// TwinCAT 3 PLC project PRG_B_StatesAndModes
// Title: B_StatesAndModes
// Company: RafalOS
// Author: Rafał Osajda
// ProjectVersion: 0.0.0.24
// ProgramVersion: 3.1.4024.0
// libraries:
//   B_Base, * (RafalOS)
//   Tc2_Standard, * (Beckhoff Automation GmbH)
//   Tc2_System, * (Beckhoff Automation GmbH)
//   Tc3_Module, * (Beckhoff Automation GmbH)
// project tree:
//   GVLs/ GVL_SaMConstans.TcGVL (not stored)
//   / PlcTask.TcTTO
//   POUs Compilation/ PRG_Compilation.TcPOU (not stored)
//   POUs/01_StatesAndModes/ E_SaMChangeCategory.TcDUT (not stored), E_SaMCommandChangeState.TcDUT, E_SaMCommandChangeMode.TcDUT (not stored), FB_SaMController.TcPOU, ITF_SaMController.TcIO, ITF_SaMControllerCommandChange.TcIO, ITF_SaMControllerConfigure.TcIO (not stored), ST_CommandChangeMode.TcDUT, ST_CommandChangeState.TcDUT, ST_SaMControllerConfigure.TcDUT (not stored), ST_SaMElementModes.TcDUT (not stored), ST_SaMElementStates.TcDUT (not stored)
//   POUs/02_CommandChange/ FB_CommandChange.TcPOU, ITF_CommandChange.TcIO (not stored)
//   POUs/03_CommandChangeState/ FB_CommandChangeAbort.TcPOU, FB_CommandChangeClear.TcPOU, FB_CommandChangeReset.TcPOU, FB_CommandChangeStart.TcPOU, FB_CommandChangeStop.TcPOU, FB_CommandChangeHold.TcPOU, FB_CommandChangeUnHold.TcPOU, FB_CommandChangeSuspend.TcPOU, FB_CommandChangeUnSuspend.TcPOU, FB_CommandChangeComplete.TcPOU
//   POUs/04_CommandChangeMode/ FB_CommandChangeProduction.TcPOU, FB_CommandChangeMaintenance.TcPOU, FB_CommandChangeManual.TcPOU, FB_CommandChangeWashing.TcPOU, FB_CommandChangeDiagnostics.TcPOU
//   POUs/05_SaMElement/ FB_SaMElement.TcPOU, ITF_SaMElement.TcIO
//   POUs/06_SaMElementStates/ FB_SaMElementAborting.TcPOU, FB_SaMElementAborted.TcPOU (not stored), FB_SaMElementUndefined.TcPOU (not stored), FB_SaMElementClearing.TcPOU (not stored), FB_SaMElementStopping.TcPOU (not stored), FB_SaMElementStopped.TcPOU, FB_SaMElementResseting.TcPOU, FB_SaMElementIdle.TcPOU (not stored), FB_SaMElementStarting.TcPOU, FB_SaMElementExecute.TcPOU (not stored), FB_SaMElementSuspending.TcPOU (not stored), FB_SaMElementSuspended.TcPOU, FB_SaMElementUnSuspending.TcPOU (not stored), FB_SaMElementHolding.TcPOU (not stored), FB_SaMElementHeld.TcPOU (not stored), FB_SaMElementUnHolding.TcPOU (not stored), FB_SaMElementCompleting.TcPOU (not stored), FB_SaMElementComplete.TcPOU (not stored)
//   POUs/07_SaMElementModes/ FB_SaMElementProduction.TcPOU, FB_SaMElementMaintenance.TcPOU (not stored), FB_SaMElementManual.TcPOU, FB_SaMElementNotAllowed.TcPOU (not stored), FB_SaMElementWashing.TcPOU, FB_SaMElementDiagnostics.TcPOU (not stored)

CONFIGURATION PRG_B_StatesAndModes
    RESOURCE PLC ON TwinCAT3
        TASK PlcTask(INTERVAL := T#10ms, PRIORITY := 20);
        PROGRAM PRG_Compilation WITH PlcTask : PRG_Compilation;
    END_RESOURCE
END_CONFIGURATION

// ---- POUs/01_StatesAndModes/E_SaMCommandChangeState.TcDUT
{attribute 'qualified_only'}
{attribute 'strict'}
TYPE E_SaMCommandChangeState :
(
	None			:= 0,
	Abort			:= 1,
    Clear			:= 2,
    Reset			:= 3,
    Start			:= 4,
    Stop			:= 5,
    Hold			:= 6,
    Unhold			:= 7,
    Suspend			:= 8,
    Unsuspend		:= 9,
    Complete		:= 10
);
END_TYPE

// ---- POUs/01_StatesAndModes/ST_CommandChangeMode.TcDUT
TYPE ST_CommandChangeMode :
STRUCT
	cmdChangeProduction	 	  	: FB_CommandChangeProduction;
	cmdChangeMaintenance		: FB_CommandChangeMaintenance;
	cmdChangeManual		    	: FB_CommandChangeManual;
	cmdChangeWashing		   	: FB_CommandChangeWashing;
	cmdChangeDiagnostics		: FB_CommandChangeDiagnostics;
END_STRUCT
END_TYPE

// ---- POUs/01_StatesAndModes/ST_CommandChangeState.TcDUT
TYPE ST_CommandChangeState :
STRUCT
	cmdChangeAbort		   		: FB_CommandChangeAbort;
	cmdChangeClear		   		: FB_CommandChangeClear;
	cmdChangeReset		   		: FB_CommandChangeReset;
	cmdChangeStart		   		: FB_CommandChangeStart;
	cmdChangeStop		    	: FB_CommandChangeStop;
	cmdChangeHold		    	: FB_CommandChangeHold;
	cmdChangeUnhold		  		: FB_CommandChangeUnHold;
	cmdChangeSuspend		 	: FB_CommandChangeSuspend;
	cmdChangeUnSuspend	  		: FB_CommandChangeUnSuspend;
	cmdChangeComplete		 	: FB_CommandChangeComplete;

END_STRUCT
END_TYPE

// ---- POUs/01_StatesAndModes/ITF_SaMController.TcIO
INTERFACE ITF_SaMController EXTENDS ITF_BaseControlElement, ITF_SaMControllerConfigure, ITF_SaMControllerCommandChange, ITF_BaseSaM

METHOD Execute : BOOL
VAR_INPUT
	iNumberOfCommand		: INT;
	eChangeCategory			: E_SaMChangeCategory;
END_VAR
END_METHOD

METHOD ExecuteTopElementOperationsForCurrentState : BOOL
VAR_INPUT
	itfTopElement				: ITF_BaseSaMStateMethod;
END_VAR
END_METHOD

METHOD PUBLIC ExitActivState
VAR_INPUT
END_VAR
END_METHOD

METHOD PUBLIC GetActiveModeName : ST_BaseLabel
VAR_INPUT
END_VAR
END_METHOD

METHOD PUBLIC GetActiveStateName : ST_BaseLabel
VAR_INPUT
END_VAR
END_METHOD

METHOD PUBLIC GetMode : E_BaseMachineMode
VAR_INPUT
END_VAR
END_METHOD

METHOD PUBLIC GetModeName : ST_BaseLabel
VAR_INPUT
	iNumber			: INT;
END_VAR
END_METHOD

METHOD PUBLIC GetState : E_BaseMachineState
VAR_INPUT
END_VAR
END_METHOD

METHOD GetStateName : ST_BaseLabel
VAR_INPUT
	iNumber			: INT;
END_VAR
END_METHOD

METHOD PUBLIC GetTimeStateForCurrentMode : LTIME
VAR_INPUT
	iNumber		: INT;
END_VAR
END_METHOD

METHOD PUBLIC GetTimeStateForMode : LTIME
VAR_INPUT
	iMode		: int;
	iState		: INT;
END_VAR
END_METHOD

METHOD PUBLIC GetTimeWorkForMode : LTIME
VAR_INPUT
	iMode	: INT;
END_VAR
END_METHOD

METHOD PUBLIC IncrementTimeStateAndMode
VAR_INPUT
	tInterval				: TIME := T#100MS;
END_VAR
END_METHOD

METHOD PUBLIC IsChangeModeBusy : BOOL
VAR_INPUT
END_VAR
END_METHOD

METHOD PUBLIC IsChangeModeDone : BOOL
VAR_INPUT
END_VAR
END_METHOD

METHOD PUBLIC IsChangeModeStatus : BOOL
VAR_INPUT
END_VAR
END_METHOD

METHOD PUBLIC IsChangeStateBusy : BOOL
VAR_INPUT
END_VAR
END_METHOD

METHOD PUBLIC IsChangeStateDone : BOOL
VAR_INPUT
END_VAR
END_METHOD

METHOD PUBLIC IsChangeStateStatus : BOOL
VAR_INPUT
END_VAR
END_METHOD

(*			
	RafalOS
	Rafał Osajda		25.11.2025		TC 4024.66
	Zwraca czy tryb o podanym numerze jest włączony
*)
METHOD IsModeEnabled : BOOL
VAR_INPUT
	iMode 	: INT;
END_VAR
END_METHOD

(*			
	RafalOS
	Rafał Osajda		25.11.2025		TC 4024.66
	Informacja czy zadany stan jest stanem aktualnym
*)
METHOD PUBLIC IsStateIsActual : BOOL
VAR_INPUT
	iTestState	: INT;
END_VAR
END_METHOD

METHOD PUBLIC IsStateTypeActive : BOOL
VAR_INPUT
END_VAR
END_METHOD

END_INTERFACE

// ---- POUs/01_StatesAndModes/ITF_SaMControllerCommandChange.TcIO
INTERFACE ITF_SaMControllerCommandChange

METHOD PUBLIC ChangeModeTo
VAR_INPUT
	eModeIn			: E_BaseMachineMode;
END_VAR
END_METHOD

METHOD PUBLIC ChangeStateTo
VAR_INPUT
	eStateIn			: E_BaseMachineState;
END_VAR
END_METHOD

METHOD PUBLIC GetState : E_BaseMachineState
VAR_INPUT
END_VAR
END_METHOD

METHOD IsModeEnebles : BOOL
VAR_INPUT
	eMode			: E_BaseMachineMode;
END_VAR
END_METHOD

METHOD IsPossibleExitActiveState : BOOL
VAR_INPUT
END_VAR
END_METHOD

METHOD IsPossibleExitState : BOOL
VAR_INPUT
	eMode		: E_BaseMachineMode;
END_VAR
END_METHOD

METHOD PUBLIC IsStateInModeEnabled : BOOL
VAR_INPUT
	eStateIn			: E_BaseMachineState;
END_VAR
END_METHOD

END_INTERFACE

// ---- POUs/05_SaMElement/ITF_SaMElement.TcIO
INTERFACE ITF_SaMElement EXTENDS ITF_BaseComponent

METHOD public GetNextState : E_BaseMachineState
VAR_INPUT
END_VAR
END_METHOD

METHOD GetTime : LTIME
VAR_INPUT
END_VAR
END_METHOD

METHOD PUBLIC IncrementTime
VAR_INPUT
	tInterval				: TIME := T#100MS;
END_VAR
END_METHOD

METHOD PUBLIC InvokeStateForTopElement : BOOL
VAR_INPUT
	itfTopElement		: ITF_BaseSaMStateMethod;
END_VAR
END_METHOD

METHOD PUBLIC IsActive : BOOL
VAR_INPUT
END_VAR
END_METHOD

(*			
	RafalOS
	Rafał Osajda		03.11.2025		TC 4024.66
	Zwraca czy element jest właczony w systemie
*)
METHOD PUBLIC IsEnabled : BOOL
VAR_INPUT
END_VAR
END_METHOD

METHOD PUBLIC IsStateTypeActive : BOOL
VAR_INPUT
END_VAR
END_METHOD

METHOD PUBLIC ResetTime
VAR_INPUT
END_VAR
END_METHOD

(*			
	RafalOS
	Rafał Osajda		03.11.2025		TC 4024.66
	Ustawia czy dane element jest aktywny
*)
METHOD PUBLIC SetActive
VAR_INPUT
	bIN			: BOOL;
END_VAR
END_METHOD

(*			
	RafalOS
	Rafał Osajda		03.11.2025		TC 4024.66
	Ustawie czy element jest włączony w systemie
*)
METHOD PUBLIC SetEnabled
VAR_INPUT
	bIN			: BOOL;
END_VAR
END_METHOD

END_INTERFACE

// ---- POUs/01_StatesAndModes/FB_SaMController.TcPOU
(*			
	RafalOS
	Rafał Osajda		30.10.2025		TC 4024.66
	Główny FB do zarządzania stanami i trybami pracy
*)
FUNCTION_BLOCK FB_SaMController EXTENDS FB_BaseControlElement IMPLEMENTS ITF_SaMController
VAR
(*	Polecenia zmiany stany	*)	
	stCmdStates					: ST_CommandChangeState;
	arrcmdStates				: ARRAY [1..GVL_SaMConstans.NUMBER_OF_COMMAND_CHANGE_STATES] OF ITF_CommandChange;
(*	Polecenia zmiany trybu	*)
	stCmdModes					: ST_CommandChangeMode;
	arrcmdModes					: ARRAY [1..GVL_SaMConstans.NUMBER_OF_COMMAND_CHANGE_MODES] OF ITF_CommandChange;
(*	Stany	*)
	arrstStates					: ARRAY [0..GVL_SaMConstans.NUMBER_OF_MODES] OF ST_SaMElementStates;
(*	Tryby	*)
	stModes						: ST_SaMElementModes;
(*	Przypisane stany do trybów	*)
	arrStatesInModes			: ARRAY [0..GVL_SaMConstans.NUMBER_OF_MODES] OF ARRAY [0..GVL_SaMConstans.NUMBER_OF_STATES] OF ITF_SaMElement;
	arrModes					: ARRAY [0..GVL_SaMConstans.NUMBER_OF_MODES] OF ITF_SaMElement;
(*	Referencja do tablicy stanów aktywnego trybu	*)
	refarrStatesForActiveMode	: REFERENCE TO ARRAY [0..GVL_SaMConstans.NUMBER_OF_STATES] OF ITF_SaMElement;
(*	Jakie trybu są aktywne	*)
	arrModeEnable				: ARRAY [0..GVL_SaMConstans.NUMBER_OF_MODES] OF BOOL;
(*	Jakie stany są aktywne w trybie	*)
	arrStateEnableInMode		: ARRAY [0..GVL_SaMConstans.NUMBER_OF_MODES] OF ARRAY [0..GVL_SaMConstans.NUMBER_OF_STATES] OF BOOL;
(*	W jakich stanach można przejść do innego trybu	*)
	arrModeTransitionEnableInState	: ARRAY [0..GVL_SaMConstans.NUMBER_OF_MODES] OF ARRAY [0..GVL_SaMConstans.NUMBER_OF_STATES] OF BOOL;
(*	Polecenia zmiany	*)
	cmdChangeMode				: FB_BaseCommand;
	cmdChangeState				: FB_BaseCommand;
(*	Zmienne		*)
	eState						: E_BaseMachineState;	//aktualny stan
	eMode						: E_BaseMachineMode;	//aktualny tryb
	eNewState					: E_BaseMachineState;	//Nowy stan
	ePrevState					: E_BaseMachineState;	//poprzedni stan
	eNewMode					: E_BaseMachineMode;	//nowy tryb
	ePrevMode					: E_BaseMachineMode;	//poprzedni tryb
END_VAR

(*			
	RafalOS
	Rafał Osajda		04.11.2025		TC 4024.66
	cykl zmiany trybu
*)
METHOD PRIVATE ChangeModeCycle : BOOL
VAR_INPUT
END_VAR
CASE THIS^.cmdChangeMode.GetStep () OF
	0	:
		THIS^.arrModes [THIS^.eMode].SetActive (bIN := FALSE);
		THIS^.ePrevMode			:= THIS^.eMode;
		THIS^.eMode				:= THIS^.eNewMode;
		THIS^.arrModes [THIS^.eMode].SetActive (bIN := TRUE);
		THIS^.refarrStatesForActiveMode	REF= THIS^.arrStatesInModes [THIS^.eMode];
		THIS^.cmdChangeMode.SetStepAsFinal ();
END_CASE
THIS^.cmdChangeMode.TestingLastCycle ();
END_METHOD

METHOD PUBLIC ChangeModeTo
VAR_INPUT
	eModeIn			: E_BaseMachineMode;
END_VAR
THIS^.eNewMode			:= eModeIn;
THIS^.cmdChangeMode.Execute ();
END_METHOD

(*			
	RafalOS
	Rafał Osajda		04.11.2025		TC 4024.66
	cykl zmiany stanu
*)
METHOD PRIVATE ChangeStateCycle : BOOL
VAR_INPUT
END_VAR
CASE THIS^.cmdChangeState.GetStep () OF
	0	:
		THIS^.refarrStatesForActiveMode [THIS^.eState].SetActive (bIN := FALSE);
		THIS^.ePrevState		:= THIS^.eState;
		THIS^.eState			:= THIS^.eNewState;
		THIS^.refarrStatesForActiveMode [THIS^.eState].SetActive (bIN := TRUE);
		THIS^.cmdChangeState.SetStepAsFinal ();
END_CASE
THIS^.cmdChangeState.TestingLastCycle ();
END_METHOD

METHOD PUBLIC ChangeStateTo
VAR_INPUT
	eStateIn			: E_BaseMachineState;
END_VAR
THIS^.eNewState			:= eStateIn;
THIS^.cmdChangeState.Execute ();
END_METHOD

(*			
	RafalOS
	Rafał Osajda		03.11.2025		TC 4024.66
	Obsługa zmiany stanów i trybów 
*)
METHOD Execute : BOOL
VAR_INPUT
	iNumberOfCommand		: INT;
	eChangeCategory			: E_SaMChangeCategory;
END_VAR
CASE eChangeCategory OF
	E_SaMChangeCategory.eState	:
		THIS^.arrcmdStates [iNumberOfCommand].Execute (iNumberOfCommand	:= iNumberOfCommand);
	E_SaMChangeCategory.eMode	:
		THIS^.arrcmdModes [iNumberOfCommand].Execute (iNumberOfCommand	:= iNumberOfCommand);
END_CASE
END_METHOD

(*			
	RafalOS
	Rafał Osajda		27.03.2025		TC 4024.66
	Obsluga bledow sprawdzanie czy jakis blad sie nei pojawil i ustawienie stanu lub wylaczenie
*)
METHOD PUBLIC ExecuteEveryCycle_Error
VAR_INPUT
END_VAR
SUPER^.ExecuteEveryCycle_Error ();
END_METHOD

(*			
	RafalOS
	Rafał Osajda		27.03.2025		TC 4024.66
	Wywolanie co cykl operacji 
*)
METHOD PUBLIC ExecuteEveryCycle_Operation
VAR_INPUT
END_VAR
SUPER^.ExecuteEveryCycle_Operation ();

IF (THIS^.cmdChangeMode.OperationExecute ()) THEN
	THIS^.cmdChangeMode.Operation (bIN := THIS^.ChangeModeCycle ());
END_IF

IF (THIS^.cmdChangeState.OperationExecute ()) THEN
	THIS^.cmdChangeState.Operation (bIN := THIS^.ChangeStateCycle ());
END_IF
END_METHOD

(*			
	RafalOS
	Rafał Osajda		27.03.2025		TC 4024.66
	Aktualizacja flag 
*)
METHOD PUBLIC ExecuteEveryCycle_Status
VAR_INST
END_VAR
SUPER^.ExecuteEveryCycle_Status ();
END_METHOD

(*			
	RafalOS
	Rafał Osajda		27.03.2025		TC 4024.66
	Testowanie czy nei pojawil sie jakis rozkaz i uruchomienie odpowiednich operacji
*)
METHOD PUBLIC ExecuteEveryCycle_Test
VAR_INPUT
END_VAR
SUPER^.ExecuteEveryCycle_Test ();

THIS^.cmdChangeMode.Test ();
THIS^.cmdChangeState.Test ();
END_METHOD

METHOD ExecuteTopElementOperationsForCurrentState : BOOL
VAR_INPUT
	itfTopElement				: ITF_BaseSaMStateMethod;
END_VAR
ExecuteTopElementOperationsForCurrentState := THIS^.refarrStatesForActiveMode [THIS^.eState].InvokeStateForTopElement (itfTopElement := itfTopElement);
END_METHOD

(*			
	RafalOS
	Rafał Osajda		04.11.2025		TC 4024.66
	Wywołanie odpowiednie metody tak by wyjśc z aktualnego stanu aktywnego 
*)
METHOD PUBLIC ExitActivState
VAR_INPUT
END_VAR
THIS^.ChangeStateTo (eStateIn := THIS^.refarrStatesForActiveMode [THIS^.eState].GetNextState ());
END_METHOD

METHOD FB_init : BOOL
VAR_INPUT
	bInitRetains : BOOL; // if TRUE, the retain variables are initialized (warm start / cold start)
	bInCopyCode : BOOL;  // if TRUE, the instance afterwards gets moved into the copy code (online change)
END_VAR
THIS^.SetText (eLocation := E_BaseLocation.pl, wsDescription := "SaM Controller");
THIS^.SetText (eLocation := E_BaseLocation.en, wsDescription := "SaM Controller");
THIS^.SetText (eLocation := E_BaseLocation.de, wsDescription := "SaM Controller");
THIS^.SetName (stName := THIS^.GetTexts ());

THIS^.Initialization_AddStates ();
THIS^.Initialization_AddModes ();

THIS^.Initialization_AddCommandChangeState ();
THIS^.Initialization_AddCommandChangeModes ();

THIS^.Initialization_StateEnabledInMode ();
THIS^.Initialization_ModeTransitionEnabledInState ();
THIS^.Initialization_ModeEnabled ();
END_METHOD

METHOD PUBLIC GetActiveModeName : ST_BaseLabel
VAR_INPUT
END_VAR
GetActiveModeName := THIS^.GetModeName (iNumber := THIS^.eMode);
END_METHOD

METHOD PUBLIC GetActiveStateName : ST_BaseLabel
VAR_INPUT
END_VAR
GetActiveStateName := THIS^.GetStateName (iNumber := THIS^.eState);
END_METHOD

METHOD PUBLIC GetMode : E_BaseMachineMode
VAR_INPUT
END_VAR
GetMode			:= THIS^.eMode;
END_METHOD

METHOD PUBLIC GetModeName : ST_BaseLabel
VAR_INPUT
	iNumber			: INT;
END_VAR
GetModeName := THIS^.arrModes [iNumber].GetName ();
END_METHOD

METHOD PUBLIC GetState : E_BaseMachineState
VAR_INPUT
END_VAR
GetState			:= THIS^.eState;
END_METHOD

METHOD GetStateName : ST_BaseLabel
VAR_INPUT
	iNumber			: INT;
END_VAR
GetStateName := THIS^.arrStatesInModes [THIS^.eMode][iNumber].GetName ();
END_METHOD

METHOD PUBLIC GetTimeStateForCurrentMode : LTIME
VAR_INPUT
	iNumber		: INT;
END_VAR
GetTimeStateForCurrentMode := this^.refarrStatesForActiveMode [iNumber].GetTime ();
END_METHOD

METHOD PUBLIC GetTimeStateForMode : LTIME
VAR_INPUT
	iMode		: INT;
	iState		: INT;
END_VAR
GetTimeStateForMode := THIS^.arrStatesInModes [iMode][iState].GetTime ();
END_METHOD

METHOD PUBLIC GetTimeWorkForMode : LTIME
VAR_INPUT
	iMode	: INT;
END_VAR
GetTimeWorkForMode := THIS^.arrModes [iMode].GetTime ();
END_METHOD

METHOD PUBLIC IncrementTimeStateAndMode
VAR_INPUT
	tInterval				: TIME := T#100MS;
END_VAR
THIS^.refarrStatesForActiveMode [THIS^.eState].IncrementTime (tInterval := tInterval);
THIS^.arrModes [THIS^.eMode].IncrementTime (tInterval := tInterval);
END_METHOD

METHOD PRIVATE Initialization_AddCommandChangeModes : BOOL
VAR_INPUT
END_VAR

THIS^.arrcmdModes [E_SaMCommandChangeMode.Production]	:= THIS^.stCmdModes.cmdChangeProduction;
THIS^.AddComponent (itfComponent 	:= THIS^.stCmdModes.cmdChangeProduction);
THIS^.stCmdModes.cmdChangeProduction.LinkSaMCotroller (itfSaMController	:= THIS^);

THIS^.arrcmdModes [E_SaMCommandChangeMode.Maintenance]	:= THIS^.stCmdModes.cmdChangeMaintenance;
THIS^.AddComponent (itfComponent 	:= THIS^.stCmdModes.cmdChangeMaintenance);
THIS^.stCmdModes.cmdChangeMaintenance.LinkSaMCotroller (itfSaMController	:= THIS^);

THIS^.arrcmdModes [E_SaMCommandChangeMode.Manual]		:= THIS^.stCmdModes.cmdChangeManual;
THIS^.AddComponent (itfComponent 	:= THIS^.stCmdModes.cmdChangeManual);
THIS^.stCmdModes.cmdChangeManual.LinkSaMCotroller (itfSaMController	:= THIS^);

THIS^.arrcmdModes [E_SaMCommandChangeMode.Washing]		:= THIS^.stCmdModes.cmdChangeWashing;
THIS^.AddComponent (itfComponent 	:= THIS^.stCmdModes.cmdChangeWashing);
THIS^.stCmdModes.cmdChangeWashing.LinkSaMCotroller (itfSaMController	:= THIS^);

THIS^.arrcmdModes [E_SaMCommandChangeMode.Diagnostisc]	:= THIS^.stCmdModes.cmdChangeDiagnostics;
THIS^.AddComponent (itfComponent 	:= THIS^.stCmdModes.cmdChangeDiagnostics);
THIS^.stCmdModes.cmdChangeDiagnostics.LinkSaMCotroller (itfSaMController	:= THIS^);
END_METHOD

METHOD PRIVATE Initialization_AddCommandChangeState : BOOL
VAR_INPUT
END_VAR
THIS^.arrcmdStates [E_SaMCommandChangeState.Abort]	:= THIS^.stCmdStates.cmdChangeAbort;
THIS^.AddComponent (itfComponent 	:= THIS^.stCmdStates.cmdChangeAbort);
THIS^.stCmdStates.cmdChangeAbort.LinkSaMCotroller (itfSaMController	:= THIS^);

THIS^.arrcmdStates [E_SaMCommandChangeState.Clear]	:= THIS^.stCmdStates.cmdChangeClear;
THIS^.AddComponent (itfComponent 	:= THIS^.stCmdStates.cmdChangeClear);
THIS^.stCmdStates.cmdChangeClear.LinkSaMCotroller (itfSaMController	:= THIS^);

THIS^.arrcmdStates [E_SaMCommandChangeState.Reset]	:= THIS^.stCmdStates.cmdChangeReset;
THIS^.AddComponent (itfComponent 	:= THIS^.stCmdStates.cmdChangeReset);
THIS^.stCmdStates.cmdChangeReset.LinkSaMCotroller (itfSaMController	:= THIS^);

THIS^.arrcmdStates [E_SaMCommandChangeState.Start]	:= THIS^.stCmdStates.cmdChangeStart;
THIS^.AddComponent (itfComponent 	:= THIS^.stCmdStates.cmdChangeStart);
THIS^.stCmdStates.cmdChangeStart.LinkSaMCotroller (itfSaMController	:= THIS^);

THIS^.arrcmdStates [E_SaMCommandChangeState.Stop]	:= THIS^.stCmdStates.cmdChangeStop;
THIS^.AddComponent (itfComponent 	:= THIS^.stCmdStates.cmdChangeStop);
THIS^.stCmdStates.cmdChangeStop.LinkSaMCotroller (itfSaMController	:= THIS^);

THIS^.arrcmdStates [E_SaMCommandChangeState.Hold]	:= THIS^.stCmdStates.cmdChangeHold;
THIS^.AddComponent (itfComponent 	:= THIS^.stCmdStates.cmdChangeHold);
THIS^.stCmdStates.cmdChangeHold.LinkSaMCotroller (itfSaMController	:= THIS^);

THIS^.arrcmdStates [E_SaMCommandChangeState.Unhold]	:= THIS^.stCmdStates.cmdChangeUnhold;
THIS^.AddComponent (itfComponent 	:= THIS^.stCmdStates.cmdChangeUnhold);
THIS^.stCmdStates.cmdChangeUnhold.LinkSaMCotroller (itfSaMController	:= THIS^);

THIS^.arrcmdStates [E_SaMCommandChangeState.Suspend]:= THIS^.stCmdStates.cmdChangeSuspend;
THIS^.AddComponent (itfComponent 	:= THIS^.stCmdStates.cmdChangeSuspend);
THIS^.stCmdStates.cmdChangeSuspend.LinkSaMCotroller (itfSaMController	:= THIS^);

THIS^.arrcmdStates [E_SaMCommandChangeState.Unsuspend]	:= THIS^.stCmdStates.cmdChangeUnSuspend;
THIS^.AddComponent (itfComponent 	:= THIS^.stCmdStates.cmdChangeUnSuspend);
THIS^.stCmdStates.cmdChangeUnSuspend.LinkSaMCotroller (itfSaMController	:= THIS^);

THIS^.arrcmdStates [E_SaMCommandChangeState.Complete]	:= THIS^.stCmdStates.cmdChangeComplete;
THIS^.AddComponent (itfComponent 	:= THIS^.stCmdStates.cmdChangeComplete);
THIS^.stCmdStates.cmdChangeComplete.LinkSaMCotroller (itfSaMController	:= THIS^);
END_METHOD

METHOD PRIVATE Initialization_AddModes : BOOL
VAR_INPUT
END_VAR
THIS^.arrModes [E_BaseMachineMode.NotAllowed]	:= THIS^.stModes.fbUndefined;
THIS^.AddComponent (itfComponent	:= THIS^.stModes.fbUndefined);
THIS^.arrModes [E_BaseMachineMode.Production]	:= THIS^.stModes.fbProduction;
THIS^.AddComponent (itfComponent	:= THIS^.stModes.fbProduction);
THIS^.arrModes [E_BaseMachineMode.Maintenance]	:= THIS^.stModes.fbMaintenance;
THIS^.AddComponent (itfComponent	:= THIS^.stModes.fbMaintenance);
THIS^.arrModes [E_BaseMachineMode.Manual]	:= THIS^.stModes.fbManual;
THIS^.AddComponent (itfComponent	:= THIS^.stModes.fbManual);
THIS^.arrModes [E_BaseMachineMode.Washing]	:= THIS^.stModes.fbWashing;
THIS^.AddComponent (itfComponent	:= THIS^.stModes.fbWashing);
THIS^.arrModes [E_BaseMachineMode.Diagnostics]	:= THIS^.stModes.fbDiagnostics;
THIS^.AddComponent (itfComponent	:= THIS^.stModes.fbDiagnostics);
END_METHOD

METHOD PRIVATE Initialization_AddStates : BOOL
VAR_INPUT
END_VAR

VAR
	iI: INT;
END_VAR
FOR iI := 0 TO GVL_SaMConstans.NUMBER_OF_MODES DO
	THIS^.arrStatesInModes [iI][E_BaseMachineState.Undefined] 		:= THIS^.arrstStates [iI].fbUndefined;
	THIS^.arrStatesInModes [iI][E_BaseMachineState.Aborting] 		:= THIS^.arrstStates [iI].fbAborting;
	THIS^.arrStatesInModes [iI][E_BaseMachineState.Aborted] 		:= THIS^.arrstStates [iI].fbAborted;
	THIS^.arrStatesInModes [iI][E_BaseMachineState.Clearing] 		:= THIS^.arrstStates [iI].fbClearing;
	THIS^.arrStatesInModes [iI][E_BaseMachineState.Stopping] 		:= THIS^.arrstStates [iI].fbStopping;
	THIS^.arrStatesInModes [iI][E_BaseMachineState.Stopped] 		:= THIS^.arrstStates [iI].fbStopped;
	THIS^.arrStatesInModes [iI][E_BaseMachineState.Resetting] 		:= THIS^.arrstStates [iI].fbResetting;
	THIS^.arrStatesInModes [iI][E_BaseMachineState.Idle] 			:= THIS^.arrstStates [iI].fbIdle;
	THIS^.arrStatesInModes [iI][E_BaseMachineState.Starting] 		:= THIS^.arrstStates [iI].fbStarting;
	THIS^.arrStatesInModes [iI][E_BaseMachineState.Execute] 		:= THIS^.arrstStates [iI].fbExecute;
	THIS^.arrStatesInModes [iI][E_BaseMachineState.Suspending]	 	:= THIS^.arrstStates [iI].fbSuspending;
	THIS^.arrStatesInModes [iI][E_BaseMachineState.Suspended] 		:= THIS^.arrstStates [iI].fbSuspended;
	THIS^.arrStatesInModes [iI][E_BaseMachineState.Unsuspending]	:= THIS^.arrstStates [iI].fbUnsuspending;
	THIS^.arrStatesInModes [iI][E_BaseMachineState.Holding] 		:= THIS^.arrstStates [iI].fbHolding;
	THIS^.arrStatesInModes [iI][E_BaseMachineState.Held] 			:= THIS^.arrstStates [iI].fbHeld;
	THIS^.arrStatesInModes [iI][E_BaseMachineState.Unholding] 		:= THIS^.arrstStates [iI].fbUnholding;
	THIS^.arrStatesInModes [iI][E_BaseMachineState.Completing] 	:= THIS^.arrstStates [iI].fbCompleting;
	THIS^.arrStatesInModes [iI][E_BaseMachineState.Complete] 		:= THIS^.arrstStates [iI].fbComplete;
	THIS^.AddComponent (itfComponent 	:= THIS^.arrstStates [iI].fbUndefined);
	THIS^.AddComponent (itfComponent 	:= THIS^.arrstStates [iI].fbAborting);
	THIS^.AddComponent (itfComponent 	:= THIS^.arrstStates [iI].fbAborted);
	THIS^.AddComponent (itfComponent 	:= THIS^.arrstStates [iI].fbClearing);
	THIS^.AddComponent (itfComponent 	:= THIS^.arrstStates [iI].fbStopping);
	THIS^.AddComponent (itfComponent 	:= THIS^.arrstStates [iI].fbStopped);
	THIS^.AddComponent (itfComponent 	:= THIS^.arrstStates [iI].fbResetting);
	THIS^.AddComponent (itfComponent 	:= THIS^.arrstStates [iI].fbIdle);
	THIS^.AddComponent (itfComponent 	:= THIS^.arrstStates [iI].fbStarting);
	THIS^.AddComponent (itfComponent 	:= THIS^.arrstStates [iI].fbExecute);
	THIS^.AddComponent (itfComponent 	:= THIS^.arrstStates [iI].fbSuspending);
	THIS^.AddComponent (itfComponent 	:= THIS^.arrstStates [iI].fbSuspended);
	THIS^.AddComponent (itfComponent 	:= THIS^.arrstStates [iI].fbUnsuspending);
	THIS^.AddComponent (itfComponent 	:= THIS^.arrstStates [iI].fbHolding);
	THIS^.AddComponent (itfComponent 	:= THIS^.arrstStates [iI].fbHeld);
	THIS^.AddComponent (itfComponent 	:= THIS^.arrstStates [iI].fbUnholding);
	THIS^.AddComponent (itfComponent 	:= THIS^.arrstStates [iI].fbCompleting);
	THIS^.AddComponent (itfComponent 	:= THIS^.arrstStates [iI].fbComplete);
END_FOR
END_METHOD

(*			
	RafalOS
	Rafał Osajda		03.11.2025		TC 4024.66
	Przepisuje ustawiony stan Enebled z elementu i zapisuje go do tablisy trybów
*)
METHOD PRIVATE Initialization_CopeEnabledMode
VAR
	iI: INT;
END_VAR
FOR iI := 0 TO GVL_SaMConstans.NUMBER_OF_MODES DO
	IF (THIS^.arrModes [iI] <> 0) THEN
		THIS^.arrModeEnable [iI]	:= THIS^.arrModes [iI].IsEnabled ();
	END_IF
END_FOR
END_METHOD

(*			
	RafalOS
	Rafał Osajda		03.11.2025		TC 4024.66
	Przepisuje ustawiony stan Enebled z elementu i zapisuje go do tablisy stanów w trybach
*)
METHOD PRIVATE Initialization_CopeEnabledStateToMode
VAR_INPUT
	eMode			: E_BaseMachineMode;
END_VAR

VAR
	iI: INT;
END_VAR
FOR iI := 0 TO GVL_SaMConstans.NUMBER_OF_STATES DO
	IF (THIS^.arrStatesInModes [eMode][iI] <> 0) THEN
		THIS^.arrStateEnableInMode [eMode][iI]	:= THIS^.arrStatesInModes [eMode][iI].IsEnabled ();
	END_IF
END_FOR
END_METHOD

(*			
	RafalOS
	Rafał Osajda		03.11.2025		TC 4024.66
	Inicjalizacja jakie tryby są właczony
*)
METHOD PRIVATE Initialization_ModeEnabled
VAR_INPUT
END_VAR
THIS^.stModes.fbUndefined.SetEnabled (bIN	:= TRUE);
THIS^.stModes.fbProduction.SetEnabled (bIN	:= TRUE);
THIS^.stModes.fbMaintenance.SetEnabled (bIN	:= TRUE);
THIS^.stModes.fbManual.SetEnabled (bIN	:= TRUE);
THIS^.stModes.fbWashing.SetEnabled (bIN	:= TRUE);
THIS^.stModes.fbDiagnostics.SetEnabled (bIN	:= TRUE);
THIS^.Initialization_CopeEnabledMode ();
END_METHOD

(*			
	RafalOS
	Rafał Osajda		03.11.2025		TC 4024.66
	Ustawienie w jakim stanie trybu mozemy zmieniać tryby
*)
METHOD PRIVATE Initialization_ModeTransitionEnabledInState
VAR_INPUT
END_VAR
THIS^.arrModeTransitionEnableInState [E_BaseMachineMode.NotAllowed][E_BaseMachineState.Undefined]		:= TRUE;
THIS^.arrModeTransitionEnableInState [E_BaseMachineMode.Production][E_BaseMachineState.Undefined]		:= TRUE;
THIS^.arrModeTransitionEnableInState [E_BaseMachineMode.Maintenance][E_BaseMachineState.Undefined]		:= TRUE;
THIS^.arrModeTransitionEnableInState [E_BaseMachineMode.Manual][E_BaseMachineState.Undefined]			:= TRUE;
THIS^.arrModeTransitionEnableInState [E_BaseMachineMode.Washing][E_BaseMachineState.Undefined]		:= TRUE;
THIS^.arrModeTransitionEnableInState [E_BaseMachineMode.Diagnostics][E_BaseMachineState.Undefined]	:= TRUE;

THIS^.arrModeTransitionEnableInState [E_BaseMachineMode.NotAllowed][E_BaseMachineState.Aborted]		:= TRUE;
THIS^.arrModeTransitionEnableInState [E_BaseMachineMode.Production][E_BaseMachineState.Aborted]		:= TRUE;
THIS^.arrModeTransitionEnableInState [E_BaseMachineMode.Maintenance][E_BaseMachineState.Aborted]		:= TRUE;
THIS^.arrModeTransitionEnableInState [E_BaseMachineMode.Manual][E_BaseMachineState.Aborted]			:= TRUE;
THIS^.arrModeTransitionEnableInState [E_BaseMachineMode.Washing][E_BaseMachineState.Aborted]			:= TRUE;
THIS^.arrModeTransitionEnableInState [E_BaseMachineMode.Diagnostics][E_BaseMachineState.Aborted]		:= TRUE;

THIS^.arrModeTransitionEnableInState [E_BaseMachineMode.NotAllowed][E_BaseMachineState.Stopped]		:= TRUE;
THIS^.arrModeTransitionEnableInState [E_BaseMachineMode.Production][E_BaseMachineState.Stopped]		:= TRUE;
THIS^.arrModeTransitionEnableInState [E_BaseMachineMode.Maintenance][E_BaseMachineState.Stopped]		:= TRUE;
THIS^.arrModeTransitionEnableInState [E_BaseMachineMode.Manual][E_BaseMachineState.Stopped]			:= TRUE;
THIS^.arrModeTransitionEnableInState [E_BaseMachineMode.Washing][E_BaseMachineState.Stopped]			:= TRUE;
THIS^.arrModeTransitionEnableInState [E_BaseMachineMode.Diagnostics][E_BaseMachineState.Stopped]		:= TRUE;
END_METHOD

(*			
	RafalOS
	Rafał Osajda		03.11.2025		TC 4024.66
	Ustawienie jakie stany sa włączone w jakim stanie
*)
METHOD PRIVATE Initialization_StateEnabledInMode
VAR_INPUT
END_VAR
THIS^.arrstStates [E_BaseMachineMode.NotAllowed].fbUndefined.SetEnabled (bIN		:= TRUE);
THIS^.arrstStates [E_BaseMachineMode.NotAllowed].fbAborting.SetEnabled (bIN		:= FALSE);
THIS^.arrstStates [E_BaseMachineMode.NotAllowed].fbAborted.SetEnabled (bIN			:= FALSE);
THIS^.arrstStates [E_BaseMachineMode.NotAllowed].fbClearing.SetEnabled (bIN 		:= FALSE);
THIS^.arrstStates [E_BaseMachineMode.NotAllowed].fbStopping.SetEnabled (bIN 		:= FALSE);
THIS^.arrstStates [E_BaseMachineMode.NotAllowed].fbStopped.SetEnabled (bIN 		:= FALSE);
THIS^.arrstStates [E_BaseMachineMode.NotAllowed].fbResetting.SetEnabled (bIN 		:= FALSE);
THIS^.arrstStates [E_BaseMachineMode.NotAllowed].fbIdle.SetEnabled (bIN 			:= FALSE);
THIS^.arrstStates [E_BaseMachineMode.NotAllowed].fbStarting.SetEnabled (bIN 		:= FALSE);
THIS^.arrstStates [E_BaseMachineMode.NotAllowed].fbExecute.SetEnabled (bIN 		:= FALSE);
THIS^.arrstStates [E_BaseMachineMode.NotAllowed].fbSuspending.SetEnabled (bIN 		:= FALSE);
THIS^.arrstStates [E_BaseMachineMode.NotAllowed].fbSuspended.SetEnabled (bIN 		:= FALSE);
THIS^.arrstStates [E_BaseMachineMode.NotAllowed].fbUnsuspending.SetEnabled (bIN	:= FALSE);
THIS^.arrstStates [E_BaseMachineMode.NotAllowed].fbHolding.SetEnabled (bIN 		:= FALSE);
THIS^.arrstStates [E_BaseMachineMode.NotAllowed].fbHeld.SetEnabled (bIN 			:= FALSE);
THIS^.arrstStates [E_BaseMachineMode.NotAllowed].fbUnholding.SetEnabled (bIN 		:= FALSE);
THIS^.arrstStates [E_BaseMachineMode.NotAllowed].fbCompleting.SetEnabled (bIN 		:= FALSE);
THIS^.arrstStates [E_BaseMachineMode.NotAllowed].fbComplete.SetEnabled (bIN 		:= FALSE);
THIS^.Initialization_CopeEnabledStateToMode (eMode	:= E_BaseMachineMode.NotAllowed);


THIS^.arrstStates [E_BaseMachineMode.Production].fbUndefined.SetEnabled (bIN		:= TRUE);
THIS^.arrstStates [E_BaseMachineMode.Production].fbAborting.SetEnabled (bIN		:= TRUE);
THIS^.arrstStates [E_BaseMachineMode.Production].fbAborted.SetEnabled (bIN			:= TRUE);
THIS^.arrstStates [E_BaseMachineMode.Production].fbClearing.SetEnabled (bIN 		:= TRUE);
THIS^.arrstStates [E_BaseMachineMode.Production].fbStopping.SetEnabled (bIN 		:= TRUE);
THIS^.arrstStates [E_BaseMachineMode.Production].fbStopped.SetEnabled (bIN 		:= TRUE);
THIS^.arrstStates [E_BaseMachineMode.Production].fbResetting.SetEnabled (bIN 		:= TRUE);
THIS^.arrstStates [E_BaseMachineMode.Production].fbIdle.SetEnabled (bIN 			:= TRUE);
THIS^.arrstStates [E_BaseMachineMode.Production].fbStarting.SetEnabled (bIN 		:= TRUE);
THIS^.arrstStates [E_BaseMachineMode.Production].fbExecute.SetEnabled (bIN 		:= TRUE);
THIS^.arrstStates [E_BaseMachineMode.Production].fbSuspending.SetEnabled (bIN 		:= TRUE);
THIS^.arrstStates [E_BaseMachineMode.Production].fbSuspended.SetEnabled (bIN 		:= TRUE);
THIS^.arrstStates [E_BaseMachineMode.Production].fbUnsuspending.SetEnabled (bIN	:= TRUE);
THIS^.arrstStates [E_BaseMachineMode.Production].fbHolding.SetEnabled (bIN 		:= TRUE);
THIS^.arrstStates [E_BaseMachineMode.Production].fbHeld.SetEnabled (bIN 			:= TRUE);
THIS^.arrstStates [E_BaseMachineMode.Production].fbUnholding.SetEnabled (bIN 		:= TRUE);
THIS^.arrstStates [E_BaseMachineMode.Production].fbCompleting.SetEnabled (bIN 		:= TRUE);
THIS^.arrstStates [E_BaseMachineMode.Production].fbComplete.SetEnabled (bIN 		:= TRUE);
THIS^.Initialization_CopeEnabledStateToMode (eMode	:= E_BaseMachineMode.Production);

THIS^.arrstStates [E_BaseMachineMode.Maintenance].fbUndefined.SetEnabled (bIN		:= TRUE);
THIS^.arrstStates [E_BaseMachineMode.Maintenance].fbAborting.SetEnabled (bIN			:= TRUE);
THIS^.arrstStates [E_BaseMachineMode.Maintenance].fbAborted.SetEnabled (bIN			:= TRUE);
THIS^.arrstStates [E_BaseMachineMode.Maintenance].fbClearing.SetEnabled (bIN 		:= TRUE);
THIS^.arrstStates [E_BaseMachineMode.Maintenance].fbStopping.SetEnabled (bIN 		:= TRUE);
THIS^.arrstStates [E_BaseMachineMode.Maintenance].fbStopped.SetEnabled (bIN 			:= TRUE);
THIS^.arrstStates [E_BaseMachineMode.Maintenance].fbResetting.SetEnabled (bIN 		:= TRUE);
THIS^.arrstStates [E_BaseMachineMode.Maintenance].fbIdle.SetEnabled (bIN 			:= TRUE);
THIS^.arrstStates [E_BaseMachineMode.Maintenance].fbStarting.SetEnabled (bIN 		:= TRUE);
THIS^.arrstStates [E_BaseMachineMode.Maintenance].fbExecute.SetEnabled (bIN 			:= TRUE);
THIS^.arrstStates [E_BaseMachineMode.Maintenance].fbSuspending.SetEnabled (bIN 		:= FALSE);
THIS^.arrstStates [E_BaseMachineMode.Maintenance].fbSuspended.SetEnabled (bIN 		:= FALSE);
THIS^.arrstStates [E_BaseMachineMode.Maintenance].fbUnsuspending.SetEnabled (bIN		:= FALSE);
THIS^.arrstStates [E_BaseMachineMode.Maintenance].fbHolding.SetEnabled (bIN 			:= FALSE);
THIS^.arrstStates [E_BaseMachineMode.Maintenance].fbHeld.SetEnabled (bIN 			:= FALSE);
THIS^.arrstStates [E_BaseMachineMode.Maintenance].fbUnholding.SetEnabled (bIN 		:= FALSE);
THIS^.arrstStates [E_BaseMachineMode.Maintenance].fbCompleting.SetEnabled (bIN 		:= FALSE);
THIS^.arrstStates [E_BaseMachineMode.Maintenance].fbComplete.SetEnabled (bIN 		:= FALSE);
THIS^.Initialization_CopeEnabledStateToMode (eMode	:= E_BaseMachineMode.Maintenance);

THIS^.arrstStates [E_BaseMachineMode.Manual].fbUndefined.SetEnabled (bIN			:= TRUE);
THIS^.arrstStates [E_BaseMachineMode.Manual].fbAborting.SetEnabled (bIN			:= TRUE);
THIS^.arrstStates [E_BaseMachineMode.Manual].fbAborted.SetEnabled (bIN				:= TRUE);
THIS^.arrstStates [E_BaseMachineMode.Manual].fbClearing.SetEnabled (bIN 			:= TRUE);
THIS^.arrstStates [E_BaseMachineMode.Manual].fbStopping.SetEnabled (bIN 			:= TRUE);
THIS^.arrstStates [E_BaseMachineMode.Manual].fbStopped.SetEnabled (bIN 			:= TRUE);
THIS^.arrstStates [E_BaseMachineMode.Manual].fbResetting.SetEnabled (bIN 			:= TRUE);
THIS^.arrstStates [E_BaseMachineMode.Manual].fbIdle.SetEnabled (bIN 				:= TRUE);
THIS^.arrstStates [E_BaseMachineMode.Manual].fbStarting.SetEnabled (bIN 			:= TRUE);
THIS^.arrstStates [E_BaseMachineMode.Manual].fbExecute.SetEnabled (bIN 			:= TRUE);
THIS^.arrstStates [E_BaseMachineMode.Manual].fbSuspending.SetEnabled (bIN 			:= TRUE);
THIS^.arrstStates [E_BaseMachineMode.Manual].fbSuspended.SetEnabled (bIN 			:= TRUE);
THIS^.arrstStates [E_BaseMachineMode.Manual].fbUnsuspending.SetEnabled (bIN		:= TRUE);
THIS^.arrstStates [E_BaseMachineMode.Manual].fbHolding.SetEnabled (bIN 			:= TRUE);
THIS^.arrstStates [E_BaseMachineMode.Manual].fbHeld.SetEnabled (bIN 				:= TRUE);
THIS^.arrstStates [E_BaseMachineMode.Manual].fbUnholding.SetEnabled (bIN 			:= TRUE);
THIS^.arrstStates [E_BaseMachineMode.Manual].fbCompleting.SetEnabled (bIN 			:= TRUE);
THIS^.arrstStates [E_BaseMachineMode.Manual].fbComplete.SetEnabled (bIN 			:= TRUE);
THIS^.Initialization_CopeEnabledStateToMode (eMode	:= E_BaseMachineMode.Manual);

THIS^.arrstStates [E_BaseMachineMode.Washing].fbUndefined.SetEnabled (bIN			:= TRUE);
THIS^.arrstStates [E_BaseMachineMode.Washing].fbAborting.SetEnabled (bIN			:= TRUE);
THIS^.arrstStates [E_BaseMachineMode.Washing].fbAborted.SetEnabled (bIN			:= TRUE);
THIS^.arrstStates [E_BaseMachineMode.Washing].fbClearing.SetEnabled (bIN 			:= TRUE);
THIS^.arrstStates [E_BaseMachineMode.Washing].fbStopping.SetEnabled (bIN 			:= TRUE);
THIS^.arrstStates [E_BaseMachineMode.Washing].fbStopped.SetEnabled (bIN 			:= TRUE);
THIS^.arrstStates [E_BaseMachineMode.Washing].fbResetting.SetEnabled (bIN 			:= TRUE);
THIS^.arrstStates [E_BaseMachineMode.Washing].fbIdle.SetEnabled (bIN 				:= TRUE);
THIS^.arrstStates [E_BaseMachineMode.Washing].fbStarting.SetEnabled (bIN 			:= TRUE);
THIS^.arrstStates [E_BaseMachineMode.Washing].fbExecute.SetEnabled (bIN 			:= TRUE);
THIS^.arrstStates [E_BaseMachineMode.Washing].fbSuspending.SetEnabled (bIN 		:= FALSE);
THIS^.arrstStates [E_BaseMachineMode.Washing].fbSuspended.SetEnabled (bIN 			:= FALSE);
THIS^.arrstStates [E_BaseMachineMode.Washing].fbUnsuspending.SetEnabled (bIN		:= FALSE);
THIS^.arrstStates [E_BaseMachineMode.Washing].fbHolding.SetEnabled (bIN 			:= FALSE);
THIS^.arrstStates [E_BaseMachineMode.Washing].fbHeld.SetEnabled (bIN 				:= FALSE);
THIS^.arrstStates [E_BaseMachineMode.Washing].fbUnholding.SetEnabled (bIN 			:= FALSE);
THIS^.arrstStates [E_BaseMachineMode.Washing].fbCompleting.SetEnabled (bIN 		:= FALSE);
THIS^.arrstStates [E_BaseMachineMode.Washing].fbComplete.SetEnabled (bIN 			:= FALSE);
THIS^.Initialization_CopeEnabledStateToMode (eMode	:= E_BaseMachineMode.Washing);

THIS^.arrstStates [E_BaseMachineMode.Diagnostics].fbUndefined.SetEnabled (bIN		:= TRUE);
THIS^.arrstStates [E_BaseMachineMode.Diagnostics].fbAborting.SetEnabled (bIN		:= TRUE);
THIS^.arrstStates [E_BaseMachineMode.Diagnostics].fbAborted.SetEnabled (bIN		:= TRUE);
THIS^.arrstStates [E_BaseMachineMode.Diagnostics].fbClearing.SetEnabled (bIN 		:= TRUE);
THIS^.arrstStates [E_BaseMachineMode.Diagnostics].fbStopping.SetEnabled (bIN 		:= TRUE);
THIS^.arrstStates [E_BaseMachineMode.Diagnostics].fbStopped.SetEnabled (bIN 		:= TRUE);
THIS^.arrstStates [E_BaseMachineMode.Diagnostics].fbResetting.SetEnabled (bIN 		:= TRUE);
THIS^.arrstStates [E_BaseMachineMode.Diagnostics].fbIdle.SetEnabled (bIN 			:= TRUE);
THIS^.arrstStates [E_BaseMachineMode.Diagnostics].fbStarting.SetEnabled (bIN 		:= TRUE);
THIS^.arrstStates [E_BaseMachineMode.Diagnostics].fbExecute.SetEnabled (bIN 		:= TRUE);
THIS^.arrstStates [E_BaseMachineMode.Diagnostics].fbSuspending.SetEnabled (bIN 	:= FALSE);
THIS^.arrstStates [E_BaseMachineMode.Diagnostics].fbSuspended.SetEnabled (bIN 		:= FALSE);
THIS^.arrstStates [E_BaseMachineMode.Diagnostics].fbUnsuspending.SetEnabled (bIN	:= FALSE);
THIS^.arrstStates [E_BaseMachineMode.Diagnostics].fbHolding.SetEnabled (bIN 		:= FALSE);
THIS^.arrstStates [E_BaseMachineMode.Diagnostics].fbHeld.SetEnabled (bIN 			:= FALSE);
THIS^.arrstStates [E_BaseMachineMode.Diagnostics].fbUnholding.SetEnabled (bIN 		:= FALSE);
THIS^.arrstStates [E_BaseMachineMode.Diagnostics].fbCompleting.SetEnabled (bIN 	:= FALSE);
THIS^.arrstStates [E_BaseMachineMode.Diagnostics].fbComplete.SetEnabled (bIN 		:= FALSE);
THIS^.Initialization_CopeEnabledStateToMode (eMode	:= E_BaseMachineMode.Diagnostics);
END_METHOD

METHOD PUBLIC IsChangeModeBusy : BOOL
VAR_INPUT
END_VAR
IsChangeModeBusy		:= THIS^.cmdChangeMode.IsBusy ();
END_METHOD

METHOD PUBLIC IsChangeModeDone : BOOL
VAR_INPUT
END_VAR
IsChangeModeDone		:= THIS^.cmdChangeMode.IsDone ();
END_METHOD

METHOD PUBLIC IsChangeModeStatus : BOOL
VAR_INPUT
END_VAR
IsChangeModeStatus		:= THIS^.cmdChangeMode.IsStatus ();
END_METHOD

METHOD PUBLIC IsChangeStateBusy : BOOL
VAR_INPUT
END_VAR
IsChangeStateBusy		:= THIS^.cmdChangeState.IsBusy ();
END_METHOD

METHOD PUBLIC IsChangeStateDone : BOOL
VAR_INPUT
END_VAR
IsChangeStateDone		:= THIS^.cmdChangeState.IsDone ();
END_METHOD

METHOD PUBLIC IsChangeStateStatus : BOOL
VAR_INPUT
END_VAR
IsChangeStateStatus		:= THIS^.cmdChangeState.IsStatus ();
END_METHOD

(*			
	RafalOS
	Rafał Osajda		25.11.2025		TC 4024.66
	Zwraca czy tryb o podanym numerze jest włączony
*)
METHOD IsModeEnabled : BOOL
VAR_INPUT
	iMode 	: INT;
END_VAR
IsModeEnabled := THIS^.arrModes [iMode].IsEnabled ();
END_METHOD

METHOD IsModeEnebles : BOOL
VAR_INPUT
	eMode			: E_BaseMachineMode;
END_VAR
IsModeEnebles		:= THIS^.arrModeEnable [eMode];
END_METHOD

METHOD IsPossibleExitActiveState : BOOL
VAR_INPUT
END_VAR
IsPossibleExitActiveState	:= THIS^.IsPossibleExitState (eMode := THIS^.eMode);
END_METHOD

METHOD IsPossibleExitState : BOOL
VAR_INPUT
	eMode		: E_BaseMachineMode;
END_VAR
IsPossibleExitState		:= THIS^.arrModeTransitionEnableInState [eMode][THIS^.eState];
END_METHOD

METHOD PUBLIC IsStateInModeEnabled : BOOL
VAR_INPUT
	eStateIn			: E_BaseMachineState;
END_VAR
IsStateInModeEnabled		:= THIS^.arrStateEnableInMode [THIS^.eMode][eStateIn];
END_METHOD

(*			
	RafalOS
	Rafał Osajda		25.11.2025		TC 4024.66
	Informacja czy zadany stan jest stanem aktualnym
*)
METHOD PUBLIC IsStateIsActual : BOOL
VAR_INPUT
	iTestState	: int;
END_VAR
IsStateIsActual := iTestState = THIS^.eState;
END_METHOD

METHOD PUBLIC IsStateTypeActive : BOOL
VAR_INPUT
END_VAR
IsStateTypeActive		:= THIS^.refarrStatesForActiveMode [THIS^.eState].IsStateTypeActive ();
END_METHOD

(*			
	RafalOS
	Rafał Osajda		03.11.2025		TC 4024.66
	Wlacza lub wylacza tryb pracy
*)
METHOD PUBLIC SetModeEnabled
VAR_INPUT
	iMode				: INT;	//numer trybu
	bValue				: BOOL;
END_VAR
THIS^.arrModes [iMode].SetEnabled (bIN	:= bValue);
THIS^.Initialization_CopeEnabledMode ();
END_METHOD

(*			
	RafalOS
	Rafał Osajda		03.11.2025		TC 4024.66
	Ustawianie czy w danym stanie może nastąpić zmiana trybu
*)
METHOD PUBLIC SetModeTransitionEnabledInState 
VAR_INPUT
	iMode			: INT;	//tryb
	iState			: INT;	//stan
	bValue			: BOOL;
END_VAR
THIS^.arrModeTransitionEnableInState [iMode][iState]	:= bValue;
END_METHOD

(*			
	RafalOS
	Rafał Osajda		03.11.2025		TC 4024.66
	Ustawia włączone stany w zadanym trybie
*)
METHOD PUBLIC SetStateEnabledInMode
VAR_INPUT
	iMode			: INT;	//tryb
	iState			: INT;	//stan
	bValue			: BOOL;
END_VAR
THIS^.arrStateEnableInMode [iMode][iState] 	:= bValue;
END_METHOD

END_FUNCTION_BLOCK

// ---- POUs/02_CommandChange/FB_CommandChange.TcPOU
FUNCTION_BLOCK ABSTRACT FB_CommandChange EXTENDS FB_BaseComponent IMPLEMENTS ITF_CommandChange
VAR
	itfSaMController				: ITF_SaMControllerCommandChange;
	
END_VAR

(*			
	RafalOS
	Rafał Osajda		24.03.2025		TC 4024.66
	Definicja nowego zgłoszenia
*)
METHOD PUBLIC EventsDefinition : BOOL
SUPER^.EventsDefinition ();
(*	1	*)
THIS^.SetText (eLocation := E_BaseLocation.pl, wsDescription	:= "Błąd przełączanie trybu - tryb docelowy jest wyłączony");
THIS^.SetText (eLocation := E_BaseLocation.en, wsDescription	:= "");
THIS^.SetText (eLocation := E_BaseLocation.de, wsDescription	:= "");
THIS^.AddEvent (
	bIgnoreRepetitions			:= FALSE,
	eEventCategory				:= E_BaseEvents_Category.Message,
	bConfirm					:= FALSE,
	stDescription				:= THIS^.GetTexts ()
);
(*	2	*)
THIS^.SetText (eLocation := E_BaseLocation.pl, wsDescription	:= "Błąd przełączanie trybu - brak możliwości wyjścia z trybu");
THIS^.SetText (eLocation := E_BaseLocation.en, wsDescription	:= "");
THIS^.SetText (eLocation := E_BaseLocation.de, wsDescription	:= "");
THIS^.AddEvent (
	bIgnoreRepetitions			:= FALSE,
	eEventCategory				:= E_BaseEvents_Category.Message,
	bConfirm					:= FALSE,
	stDescription				:= THIS^.GetTexts ()
);
(*	3	*)
THIS^.SetText (eLocation := E_BaseLocation.pl, wsDescription	:= "Błąd przełączanie trybu - brak możliwości wejścia do trybu");
THIS^.SetText (eLocation := E_BaseLocation.en, wsDescription	:= "");
THIS^.SetText (eLocation := E_BaseLocation.de, wsDescription	:= "");
THIS^.AddEvent (
	bIgnoreRepetitions			:= FALSE,
	eEventCategory				:= E_BaseEvents_Category.Message,
	bConfirm					:= FALSE,
	stDescription				:= THIS^.GetTexts ()
);
(*	4	*)
THIS^.SetText (eLocation := E_BaseLocation.pl, wsDescription	:= "Błąd przełączanie stanu - te polecenie nie obsługuje tego stanu");
THIS^.SetText (eLocation := E_BaseLocation.en, wsDescription	:= "");
THIS^.SetText (eLocation := E_BaseLocation.de, wsDescription	:= "");
THIS^.AddEvent (
	bIgnoreRepetitions			:= FALSE,
	eEventCategory				:= E_BaseEvents_Category.Message,
	bConfirm					:= FALSE,
	stDescription				:= THIS^.GetTexts ()
);
(*	5	*)
THIS^.SetText (eLocation := E_BaseLocation.pl, wsDescription	:= "Błąd przełączanie stanu - decelowy stan jest wyłączony");
THIS^.SetText (eLocation := E_BaseLocation.en, wsDescription	:= "");
THIS^.SetText (eLocation := E_BaseLocation.de, wsDescription	:= "");
THIS^.AddEvent (
	bIgnoreRepetitions			:= FALSE,
	eEventCategory				:= E_BaseEvents_Category.Message,
	bConfirm					:= FALSE,
	stDescription				:= THIS^.GetTexts ()
);
END_METHOD

(*			
	RafalOS
	Rafał Osajda		03.11.2025		TC 4024.66
	Test czy można zmienić stan lub tryb i zwraca czy można i uruchamia zmianę
*)
METHOD PUBLIC Execute : BOOL
VAR_INPUT
	iNumberOfCommand	: INT;
END_VAR
END_METHOD

(*			
	RafalOS
	Rafał Osajda		03.11.2025		TC 4024.66
	Podłączenie sterowania do SaMController
*)
METHOD PUBLIC LinkSaMCotroller : BOOL
VAR_INPUT
	itfSaMController		: ITF_SaMControllerCommandChange;
END_VAR
THIS^.itfSaMController		:= itfSaMController;
END_METHOD

END_FUNCTION_BLOCK

// ---- POUs/03_CommandChangeState/FB_CommandChangeAbort.TcPOU
FUNCTION_BLOCK FB_CommandChangeAbort EXTENDS FB_CommandChange IMPLEMENTS ITF_CommandChange
VAR

END_VAR

(*			
	RafalOS
	Rafał Osajda		03.11.2025		TC 4024.66
	Test czy można zmienić stan lub tryb i zwraca czy można i uruchamia zmianę
*)
METHOD PUBLIC Execute : BOOL
VAR_INPUT
	iNumberOfCommand	: INT;
END_VAR
IF (THIS^.itfSaMController.GetState () = E_BaseMachineState.Resetting OR
	THIS^.itfSaMController.GetState () = E_BaseMachineState.Idle OR
	THIS^.itfSaMController.GetState () = E_BaseMachineState.Starting OR
	THIS^.itfSaMController.GetState () = E_BaseMachineState.Execute OR
	THIS^.itfSaMController.GetState () = E_BaseMachineState.Suspending OR
	THIS^.itfSaMController.GetState () = E_BaseMachineState.Suspended OR
	THIS^.itfSaMController.GetState () = E_BaseMachineState.Unsuspending OR
	THIS^.itfSaMController.GetState () = E_BaseMachineState.Holding OR
	THIS^.itfSaMController.GetState () = E_BaseMachineState.Held OR
	THIS^.itfSaMController.GetState () = E_BaseMachineState.Unholding OR
	THIS^.itfSaMController.GetState () = E_BaseMachineState.Completing OR
	THIS^.itfSaMController.GetState () = E_BaseMachineState.Complete OR
	THIS^.itfSaMController.GetState () = E_BaseMachineState.Stopped OR
	THIS^.itfSaMController.GetState () = E_BaseMachineState.Stopping OR
	THIS^.itfSaMController.GetState () = E_BaseMachineState.Clearing OR
	THIS^.itfSaMController.GetState () = E_BaseMachineState.Undefined) THEN		// sprawdzenie czy jesteśmy w dobrym stanie dla tego rozkazu
	IF (THIS^.itfSaMController.IsStateInModeEnabled (eStateIn := E_BaseMachineState.Aborting)) THEN	//test czy stan do którego chcemy przejśc jest właczony dla tego trybu
		THIS^.itfSaMController.ChangeStateTo (eStateIn := E_BaseMachineState.Aborting);
	ELSE
		THIS^.EventSetActive (iNumber := 5);	//stan docelowy jest wylaczony w tym trybie
	END_IF
ELSE
	THIS^.EventSetActive (iNumber := 4);	//ten rozkaz nie obsluguje tego stanu
END_IF
END_METHOD

METHOD FB_init : BOOL
VAR_INPUT
	bInitRetains : BOOL; // if TRUE, the retain variables are initialized (warm start / cold start)
	bInCopyCode : BOOL;  // if TRUE, the instance afterwards gets moved into the copy code (online change)
END_VAR
THIS^.SetText (eLocation := E_BaseLocation.pl, wsDescription := "Command change state - Abort");
THIS^.SetText (eLocation := E_BaseLocation.en, wsDescription := "Command change state - Abort");
THIS^.SetText (eLocation := E_BaseLocation.de, wsDescription := "Command change state - Abort");
THIS^.SetName (stName := THIS^.GetTexts ());
END_METHOD

END_FUNCTION_BLOCK

// ---- POUs/03_CommandChangeState/FB_CommandChangeClear.TcPOU
FUNCTION_BLOCK FB_CommandChangeClear EXTENDS FB_CommandChange IMPLEMENTS ITF_CommandChange
VAR

END_VAR

(*			
	RafalOS
	Rafał Osajda		03.11.2025		TC 4024.66
	Test czy można zmienić stan lub tryb i zwraca czy można i uruchamia zmianę
*)
METHOD PUBLIC Execute : BOOL
VAR_INPUT
	iNumberOfCommand	: INT;
END_VAR
IF (THIS^.itfSaMController.GetState () = E_BaseMachineState.Aborted) THEN		// sprawdzenie czy jesteśmy w dobrym stanie dla tego rozkazu
	IF (THIS^.itfSaMController.IsStateInModeEnabled (eStateIn := E_BaseMachineState.Clearing)) THEN	//test czy stan do którego chcemy przejśc jest właczony dla tego trybu
		THIS^.itfSaMController.ChangeStateTo (eStateIn := E_BaseMachineState.Clearing);
	ELSE
		THIS^.EventSetActive (iNumber := 5);	//stan docelowy jest wylaczony w tym trybie
	END_IF
ELSE
	THIS^.EventSetActive (iNumber := 4);	//ten rozkaz nie obsluguje tego stanu
END_IF
END_METHOD

METHOD FB_init : BOOL
VAR_INPUT
	bInitRetains : BOOL; // if TRUE, the retain variables are initialized (warm start / cold start)
	bInCopyCode : BOOL;  // if TRUE, the instance afterwards gets moved into the copy code (online change)
END_VAR
THIS^.SetText (eLocation := E_BaseLocation.pl, wsDescription := "Command change state - Clear");
THIS^.SetText (eLocation := E_BaseLocation.en, wsDescription := "Command change state - Clear");
THIS^.SetText (eLocation := E_BaseLocation.de, wsDescription := "Command change state - Clear");
THIS^.SetName (stName := THIS^.GetTexts ());
END_METHOD

END_FUNCTION_BLOCK

// ---- POUs/03_CommandChangeState/FB_CommandChangeReset.TcPOU
FUNCTION_BLOCK FB_CommandChangeReset EXTENDS FB_CommandChange IMPLEMENTS ITF_CommandChange
VAR

END_VAR

(*			
	RafalOS
	Rafał Osajda		03.11.2025		TC 4024.66
	Test czy można zmienić stan lub tryb i zwraca czy można i uruchamia zmianę
*)
METHOD PUBLIC Execute : BOOL
VAR_INPUT
	iNumberOfCommand	: INT;
END_VAR
IF (THIS^.itfSaMController.GetState () = E_BaseMachineState.Stopped OR
	THIS^.itfSaMController.GetState () = E_BaseMachineState.Complete) THEN		// sprawdzenie czy jesteśmy w dobrym stanie dla tego rozkazu
	IF (THIS^.itfSaMController.IsStateInModeEnabled (eStateIn := E_BaseMachineState.Resetting)) THEN	//test czy stan do którego chcemy przejśc jest właczony dla tego trybu
		THIS^.itfSaMController.ChangeStateTo (eStateIn := E_BaseMachineState.Resetting);
	ELSE
		THIS^.EventSetActive (iNumber := 5);	//stan docelowy jest wylaczony w tym trybie
	END_IF
ELSE
	THIS^.EventSetActive (iNumber := 4);	//ten rozkaz nie obsluguje tego stanu
END_IF
END_METHOD

METHOD FB_init : BOOL
VAR_INPUT
	bInitRetains : BOOL; // if TRUE, the retain variables are initialized (warm start / cold start)
	bInCopyCode : BOOL;  // if TRUE, the instance afterwards gets moved into the copy code (online change)
END_VAR
THIS^.SetText (eLocation := E_BaseLocation.pl, wsDescription := "Command change state - Reset");
THIS^.SetText (eLocation := E_BaseLocation.en, wsDescription := "Command change state - Reset");
THIS^.SetText (eLocation := E_BaseLocation.de, wsDescription := "Command change state - Reset");
THIS^.SetName (stName := THIS^.GetTexts ());
END_METHOD

END_FUNCTION_BLOCK

// ---- POUs/03_CommandChangeState/FB_CommandChangeStart.TcPOU
FUNCTION_BLOCK FB_CommandChangeStart EXTENDS FB_CommandChange IMPLEMENTS ITF_CommandChange
VAR

END_VAR

(*			
	RafalOS
	Rafał Osajda		03.11.2025		TC 4024.66
	Test czy można zmienić stan lub tryb i zwraca czy można i uruchamia zmianę
*)
METHOD PUBLIC Execute : BOOL
VAR_INPUT
	iNumberOfCommand	: INT;
END_VAR
IF (THIS^.itfSaMController.GetState () = E_BaseMachineState.Idle) THEN		// sprawdzenie czy jesteśmy w dobrym stanie dla tego rozkazu
	IF (THIS^.itfSaMController.IsStateInModeEnabled (eStateIn := E_BaseMachineState.Starting)) THEN	//test czy stan do którego chcemy przejśc jest właczony dla tego trybu
		THIS^.itfSaMController.ChangeStateTo (eStateIn := E_BaseMachineState.Starting);
	ELSE
		THIS^.EventSetActive (iNumber := 5);	//stan docelowy jest wylaczony w tym trybie
	END_IF
ELSE
	THIS^.EventSetActive (iNumber := 4);	//ten rozkaz nie obsluguje tego stanu
END_IF
END_METHOD

METHOD FB_init : BOOL
VAR_INPUT
	bInitRetains : BOOL; // if TRUE, the retain variables are initialized (warm start / cold start)
	bInCopyCode : BOOL;  // if TRUE, the instance afterwards gets moved into the copy code (online change)
END_VAR
THIS^.SetText (eLocation := E_BaseLocation.pl, wsDescription := "Command change state - Start");
THIS^.SetText (eLocation := E_BaseLocation.en, wsDescription := "Command change state - Start");
THIS^.SetText (eLocation := E_BaseLocation.de, wsDescription := "Command change state - Start");
THIS^.SetName (stName := THIS^.GetTexts ());
END_METHOD

END_FUNCTION_BLOCK

// ---- POUs/03_CommandChangeState/FB_CommandChangeStop.TcPOU
FUNCTION_BLOCK FB_CommandChangeStop EXTENDS FB_CommandChange IMPLEMENTS ITF_CommandChange
VAR

END_VAR

(*			
	RafalOS
	Rafał Osajda		03.11.2025		TC 4024.66
	Test czy można zmienić stan lub tryb i zwraca czy można i uruchamia zmianę
*)
METHOD PUBLIC Execute : BOOL
VAR_INPUT
	iNumberOfCommand	: INT;
END_VAR
IF (THIS^.itfSaMController.GetState () = E_BaseMachineState.Resetting OR
	THIS^.itfSaMController.GetState () = E_BaseMachineState.Idle OR
	THIS^.itfSaMController.GetState () = E_BaseMachineState.Starting OR
	THIS^.itfSaMController.GetState () = E_BaseMachineState.Execute OR
	THIS^.itfSaMController.GetState () = E_BaseMachineState.Suspending OR
	THIS^.itfSaMController.GetState () = E_BaseMachineState.Suspended OR
	THIS^.itfSaMController.GetState () = E_BaseMachineState.Unsuspending OR
	THIS^.itfSaMController.GetState () = E_BaseMachineState.Holding OR
	THIS^.itfSaMController.GetState () = E_BaseMachineState.Held OR
	THIS^.itfSaMController.GetState () = E_BaseMachineState.Unholding OR
	THIS^.itfSaMController.GetState () = E_BaseMachineState.Completing OR
	THIS^.itfSaMController.GetState () = E_BaseMachineState.Complete) THEN		// sprawdzenie czy jesteśmy w dobrym stanie dla tego rozkazu
	IF (THIS^.itfSaMController.IsStateInModeEnabled (eStateIn := E_BaseMachineState.Stopping)) THEN	//test czy stan do którego chcemy przejśc jest właczony dla tego trybu
		THIS^.itfSaMController.ChangeStateTo (eStateIn := E_BaseMachineState.Stopping);
	ELSE
		THIS^.EventSetActive (iNumber := 5);	//stan docelowy jest wylaczony w tym trybie
	END_IF
ELSE
	THIS^.EventSetActive (iNumber := 4);	//ten rozkaz nie obsluguje tego stanu
END_IF
END_METHOD

METHOD FB_init : BOOL
VAR_INPUT
	bInitRetains : BOOL; // if TRUE, the retain variables are initialized (warm start / cold start)
	bInCopyCode : BOOL;  // if TRUE, the instance afterwards gets moved into the copy code (online change)
END_VAR
THIS^.SetText (eLocation := E_BaseLocation.pl, wsDescription := "Command change state - Stop");
THIS^.SetText (eLocation := E_BaseLocation.en, wsDescription := "Command change state - Stop");
THIS^.SetText (eLocation := E_BaseLocation.de, wsDescription := "Command change state - Stop");
THIS^.SetName (stName := THIS^.GetTexts ());
END_METHOD

END_FUNCTION_BLOCK

// ---- POUs/03_CommandChangeState/FB_CommandChangeHold.TcPOU
FUNCTION_BLOCK FB_CommandChangeHold EXTENDS FB_CommandChange IMPLEMENTS ITF_CommandChange
VAR

END_VAR

(*			
	RafalOS
	Rafał Osajda		03.11.2025		TC 4024.66
	Test czy można zmienić stan lub tryb i zwraca czy można i uruchamia zmianę
*)
METHOD PUBLIC Execute : BOOL
VAR_INPUT
	iNumberOfCommand	: INT;
END_VAR
IF (THIS^.itfSaMController.GetState () = E_BaseMachineState.Execute) THEN		// sprawdzenie czy jesteśmy w dobrym stanie dla tego rozkazu
	IF (THIS^.itfSaMController.IsStateInModeEnabled (eStateIn := E_BaseMachineState.Holding)) THEN	//test czy stan do którego chcemy przejśc jest właczony dla tego trybu
		THIS^.itfSaMController.ChangeStateTo (eStateIn := E_BaseMachineState.Holding);
	ELSE
		THIS^.EventSetActive (iNumber := 5);	//stan docelowy jest wylaczony w tym trybie
	END_IF
ELSE
	THIS^.EventSetActive (iNumber := 4);	//ten rozkaz nie obsluguje tego stanu
END_IF
END_METHOD

METHOD FB_init : BOOL
VAR_INPUT
	bInitRetains : BOOL; // if TRUE, the retain variables are initialized (warm start / cold start)
	bInCopyCode : BOOL;  // if TRUE, the instance afterwards gets moved into the copy code (online change)
END_VAR
THIS^.SetText (eLocation := E_BaseLocation.pl, wsDescription := "Command change state - Hold");
THIS^.SetText (eLocation := E_BaseLocation.en, wsDescription := "Command change state - Hold");
THIS^.SetText (eLocation := E_BaseLocation.de, wsDescription := "Command change state - Hold");
THIS^.SetName (stName := THIS^.GetTexts ());
END_METHOD

END_FUNCTION_BLOCK

// ---- POUs/03_CommandChangeState/FB_CommandChangeUnHold.TcPOU
FUNCTION_BLOCK FB_CommandChangeUnHold EXTENDS FB_CommandChange IMPLEMENTS ITF_CommandChange
VAR

END_VAR

(*			
	RafalOS
	Rafał Osajda		03.11.2025		TC 4024.66
	Test czy można zmienić stan lub tryb i zwraca czy można i uruchamia zmianę
*)
METHOD PUBLIC Execute : BOOL
VAR_INPUT
	iNumberOfCommand	: INT;
END_VAR
IF (THIS^.itfSaMController.GetState () = E_BaseMachineState.Held) THEN		// sprawdzenie czy jesteśmy w dobrym stanie dla tego rozkazu
	IF (THIS^.itfSaMController.IsStateInModeEnabled (eStateIn := E_BaseMachineState.Unholding)) THEN	//test czy stan do którego chcemy przejśc jest właczony dla tego trybu
		THIS^.itfSaMController.ChangeStateTo (eStateIn := E_BaseMachineState.Unholding);
	ELSE
		THIS^.EventSetActive (iNumber := 5);	//stan docelowy jest wylaczony w tym trybie
	END_IF
ELSE
	THIS^.EventSetActive (iNumber := 4);	//ten rozkaz nie obsluguje tego stanu
END_IF
END_METHOD

METHOD FB_init : BOOL
VAR_INPUT
	bInitRetains : BOOL; // if TRUE, the retain variables are initialized (warm start / cold start)
	bInCopyCode : BOOL;  // if TRUE, the instance afterwards gets moved into the copy code (online change)
END_VAR
THIS^.SetText (eLocation := E_BaseLocation.pl, wsDescription := "Command change state - UnHold");
THIS^.SetText (eLocation := E_BaseLocation.en, wsDescription := "Command change state - UnHold");
THIS^.SetText (eLocation := E_BaseLocation.de, wsDescription := "Command change state - UnHold");
THIS^.SetName (stName := THIS^.GetTexts ());
END_METHOD

END_FUNCTION_BLOCK

// ---- POUs/03_CommandChangeState/FB_CommandChangeSuspend.TcPOU
FUNCTION_BLOCK FB_CommandChangeSuspend EXTENDS FB_CommandChange IMPLEMENTS ITF_CommandChange
VAR

END_VAR

(*			
	RafalOS
	Rafał Osajda		03.11.2025		TC 4024.66
	Test czy można zmienić stan lub tryb i zwraca czy można i uruchamia zmianę
*)
METHOD PUBLIC Execute : BOOL
VAR_INPUT
	iNumberOfCommand	: INT;
END_VAR
IF (THIS^.itfSaMController.GetState () = E_BaseMachineState.Execute) THEN		// sprawdzenie czy jesteśmy w dobrym stanie dla tego rozkazu
	IF (THIS^.itfSaMController.IsStateInModeEnabled (eStateIn := E_BaseMachineState.Suspending)) THEN	//test czy stan do którego chcemy przejśc jest właczony dla tego trybu
		THIS^.itfSaMController.ChangeStateTo (eStateIn := E_BaseMachineState.Suspending);
	ELSE
		THIS^.EventSetActive (iNumber := 5);	//stan docelowy jest wylaczony w tym trybie
	END_IF
ELSE
	THIS^.EventSetActive (iNumber := 4);	//ten rozkaz nie obsluguje tego stanu
END_IF
END_METHOD

METHOD FB_init : BOOL
VAR_INPUT
	bInitRetains : BOOL; // if TRUE, the retain variables are initialized (warm start / cold start)
	bInCopyCode : BOOL;  // if TRUE, the instance afterwards gets moved into the copy code (online change)
END_VAR
THIS^.SetText (eLocation := E_BaseLocation.pl, wsDescription := "Command change state - Suspend");
THIS^.SetText (eLocation := E_BaseLocation.en, wsDescription := "Command change state - Suspend");
THIS^.SetText (eLocation := E_BaseLocation.de, wsDescription := "Command change state - Suspend");
THIS^.SetName (stName := THIS^.GetTexts ());
END_METHOD

END_FUNCTION_BLOCK

// ---- POUs/03_CommandChangeState/FB_CommandChangeUnSuspend.TcPOU
FUNCTION_BLOCK FB_CommandChangeUnSuspend EXTENDS FB_CommandChange IMPLEMENTS ITF_CommandChange
VAR

END_VAR

(*			
	RafalOS
	Rafał Osajda		03.11.2025		TC 4024.66
	Test czy można zmienić stan lub tryb i zwraca czy można i uruchamia zmianę
*)
METHOD PUBLIC Execute : BOOL
VAR_INPUT
	iNumberOfCommand	: INT;
END_VAR
IF (THIS^.itfSaMController.GetState () = E_BaseMachineState.Suspended) THEN		// sprawdzenie czy jesteśmy w dobrym stanie dla tego rozkazu
	IF (THIS^.itfSaMController.IsStateInModeEnabled (eStateIn := E_BaseMachineState.Unsuspending)) THEN	//test czy stan do którego chcemy przejśc jest właczony dla tego trybu
		THIS^.itfSaMController.ChangeStateTo (eStateIn := E_BaseMachineState.Unsuspending);
	ELSE
		THIS^.EventSetActive (iNumber := 5);	//stan docelowy jest wylaczony w tym trybie
	END_IF
ELSE
	THIS^.EventSetActive (iNumber := 4);	//ten rozkaz nie obsluguje tego stanu
END_IF
END_METHOD

METHOD FB_init : BOOL
VAR_INPUT
	bInitRetains : BOOL; // if TRUE, the retain variables are initialized (warm start / cold start)
	bInCopyCode : BOOL;  // if TRUE, the instance afterwards gets moved into the copy code (online change)
END_VAR
THIS^.SetText (eLocation := E_BaseLocation.pl, wsDescription := "Command change state - UnSuspend");
THIS^.SetText (eLocation := E_BaseLocation.en, wsDescription := "Command change state - UnSuspend");
THIS^.SetText (eLocation := E_BaseLocation.de, wsDescription := "Command change state - UnSuspend");
THIS^.SetName (stName := THIS^.GetTexts ());
END_METHOD

END_FUNCTION_BLOCK

// ---- POUs/03_CommandChangeState/FB_CommandChangeComplete.TcPOU
FUNCTION_BLOCK FB_CommandChangeComplete EXTENDS FB_CommandChange  IMPLEMENTS ITF_CommandChange
VAR

END_VAR

(*			
	RafalOS
	Rafał Osajda		03.11.2025		TC 4024.66
	Test czy można zmienić stan lub tryb i zwraca czy można i uruchamia zmianę
*)
METHOD PUBLIC Execute : BOOL
VAR_INPUT
	iNumberOfCommand	: INT;
END_VAR
IF (THIS^.itfSaMController.GetState () = E_BaseMachineState.Execute) THEN		// sprawdzenie czy jesteśmy w dobrym stanie dla tego rozkazu
	IF (THIS^.itfSaMController.IsStateInModeEnabled (eStateIn := E_BaseMachineState.Completing)) THEN	//test czy stan do którego chcemy przejśc jest właczony dla tego trybu
		THIS^.itfSaMController.ChangeStateTo (eStateIn := E_BaseMachineState.Completing);
	ELSE
		THIS^.EventSetActive (iNumber := 5);	//stan docelowy jest wylaczony w tym trybie
	END_IF
ELSE
	THIS^.EventSetActive (iNumber := 4);	//ten rozkaz nie obsluguje tego stanu
END_IF
END_METHOD

METHOD FB_init : BOOL
VAR_INPUT
	bInitRetains : BOOL; // if TRUE, the retain variables are initialized (warm start / cold start)
	bInCopyCode : BOOL;  // if TRUE, the instance afterwards gets moved into the copy code (online change)
END_VAR
THIS^.SetText (eLocation := E_BaseLocation.pl, wsDescription := "Command change state - Complete");
THIS^.SetText (eLocation := E_BaseLocation.en, wsDescription := "Command change state - Complete");
THIS^.SetText (eLocation := E_BaseLocation.de, wsDescription := "Command change state - Complete");
THIS^.SetName (stName := THIS^.GetTexts ());
END_METHOD

END_FUNCTION_BLOCK

// ---- POUs/04_CommandChangeMode/FB_CommandChangeProduction.TcPOU
FUNCTION_BLOCK FB_CommandChangeProduction EXTENDS FB_CommandChange IMPLEMENTS ITF_CommandChange
VAR

END_VAR

(*			
	RafalOS
	Rafał Osajda		03.11.2025		TC 4024.66
	Test czy można zmienić stan lub tryb i zwraca czy można i uruchamia zmianę
*)
METHOD PUBLIC Execute : BOOL
VAR_INPUT
	iNumberOfCommand	: INT;
END_VAR
IF (THIS^.itfSaMController.IsModeEnebles (eMode := E_BaseMachineMode.Production)) THEN
	IF (THIS^.itfSaMController.IsPossibleExitActiveState ()) THEN
		IF (THIS^.itfSaMController.IsPossibleExitState (eMode := E_BaseMachineMode.Production)) THEN
			THIS^.itfSaMController.ChangeModeTo (eModeIn := E_BaseMachineMode.Production);
		ELSE
			THIS^.EventSetActive (iNumber := 3);	//brak możlwiosći wejście do trybu w tym stanie 
		END_IF
	ELSE
		THIS^.EventSetActive (iNumber := 2);	//brak możliwości wyjścia w tym stanie z tego trybu
	END_IF
ELSE
	THIS^.EventSetActive (iNumber := 1);	//tryb docelowy wylaczony
END_IF
END_METHOD

METHOD FB_init : BOOL
VAR_INPUT
	bInitRetains : BOOL; // if TRUE, the retain variables are initialized (warm start / cold start)
	bInCopyCode : BOOL;  // if TRUE, the instance afterwards gets moved into the copy code (online change)
END_VAR
THIS^.SetText (eLocation := E_BaseLocation.pl, wsDescription := "Command change mode - Production");
THIS^.SetText (eLocation := E_BaseLocation.en, wsDescription := "Command change mode - Production");
THIS^.SetText (eLocation := E_BaseLocation.de, wsDescription := "Command change mode - Production");
THIS^.SetName (stName := THIS^.GetTexts ());
END_METHOD

END_FUNCTION_BLOCK

// ---- POUs/04_CommandChangeMode/FB_CommandChangeMaintenance.TcPOU
FUNCTION_BLOCK FB_CommandChangeMaintenance EXTENDS FB_CommandChange IMPLEMENTS ITF_CommandChange
VAR

END_VAR

(*			
	RafalOS
	Rafał Osajda		03.11.2025		TC 4024.66
	Test czy można zmienić stan lub tryb i zwraca czy można i uruchamia zmianę
*)
METHOD PUBLIC Execute : BOOL
VAR_INPUT
	iNumberOfCommand	: INT;
END_VAR
IF (THIS^.itfSaMController.IsModeEnebles (eMode := E_BaseMachineMode.Maintenance)) THEN
	IF (THIS^.itfSaMController.IsPossibleExitActiveState ()) THEN
		IF (THIS^.itfSaMController.IsPossibleExitState (eMode := E_BaseMachineMode.Maintenance)) THEN
			THIS^.itfSaMController.ChangeModeTo (eModeIn := E_BaseMachineMode.Maintenance);
		ELSE
			THIS^.EventSetActive (iNumber := 3);	//brak możlwiosći wejście do trybu w tym stanie 
		END_IF
	ELSE
		THIS^.EventSetActive (iNumber := 2);	//brak możliwości wyjścia w tym stanie z tego trybu
	END_IF
ELSE
	THIS^.EventSetActive (iNumber := 1);	//tryb docelowy wylaczony
END_IF
END_METHOD

METHOD FB_init : BOOL
VAR_INPUT
	bInitRetains : BOOL; // if TRUE, the retain variables are initialized (warm start / cold start)
	bInCopyCode : BOOL;  // if TRUE, the instance afterwards gets moved into the copy code (online change)
END_VAR
THIS^.SetText (eLocation := E_BaseLocation.pl, wsDescription := "Command change mode - Maintenance");
THIS^.SetText (eLocation := E_BaseLocation.en, wsDescription := "Command change mode - Maintenance");
THIS^.SetText (eLocation := E_BaseLocation.de, wsDescription := "Command change mode - Maintenance");
THIS^.SetName (stName := THIS^.GetTexts ());
END_METHOD

END_FUNCTION_BLOCK

// ---- POUs/04_CommandChangeMode/FB_CommandChangeManual.TcPOU
FUNCTION_BLOCK FB_CommandChangeManual EXTENDS FB_CommandChange IMPLEMENTS ITF_CommandChange
VAR

END_VAR

(*			
	RafalOS
	Rafał Osajda		03.11.2025		TC 4024.66
	Test czy można zmienić stan lub tryb i zwraca czy można i uruchamia zmianę
*)
METHOD PUBLIC Execute : BOOL
VAR_INPUT
	iNumberOfCommand	: INT;
END_VAR
IF (THIS^.itfSaMController.IsModeEnebles (eMode := E_BaseMachineMode.Manual)) THEN
	IF (THIS^.itfSaMController.IsPossibleExitActiveState ()) THEN
		IF (THIS^.itfSaMController.IsPossibleExitState (eMode := E_BaseMachineMode.Manual)) THEN
			THIS^.itfSaMController.ChangeModeTo (eModeIn := E_BaseMachineMode.Manual);
		ELSE
			THIS^.EventSetActive (iNumber := 3);	//brak możlwiosći wejście do trybu w tym stanie 
		END_IF
	ELSE
		THIS^.EventSetActive (iNumber := 2);	//brak możliwości wyjścia w tym stanie z tego trybu
	END_IF
ELSE
	THIS^.EventSetActive (iNumber := 1);	//tryb docelowy wylaczony
END_IF
END_METHOD

METHOD FB_init : BOOL
VAR_INPUT
	bInitRetains : BOOL; // if TRUE, the retain variables are initialized (warm start / cold start)
	bInCopyCode : BOOL;  // if TRUE, the instance afterwards gets moved into the copy code (online change)
END_VAR
THIS^.SetText (eLocation := E_BaseLocation.pl, wsDescription := "Command change mode - Manual");
THIS^.SetText (eLocation := E_BaseLocation.en, wsDescription := "Command change mode - Manual");
THIS^.SetText (eLocation := E_BaseLocation.de, wsDescription := "Command change mode - Manual");
THIS^.SetName (stName := THIS^.GetTexts ());
END_METHOD

END_FUNCTION_BLOCK

// ---- POUs/04_CommandChangeMode/FB_CommandChangeWashing.TcPOU
FUNCTION_BLOCK FB_CommandChangeWashing EXTENDS FB_CommandChange IMPLEMENTS ITF_CommandChange
VAR

END_VAR

(*			
	RafalOS
	Rafał Osajda		03.11.2025		TC 4024.66
	Test czy można zmienić stan lub tryb i zwraca czy można i uruchamia zmianę
*)
METHOD PUBLIC Execute : BOOL
VAR_INPUT
	iNumberOfCommand	: INT;
END_VAR
IF (THIS^.itfSaMController.IsModeEnebles (eMode := E_BaseMachineMode.Washing)) THEN
	IF (THIS^.itfSaMController.IsPossibleExitActiveState ()) THEN
		IF (THIS^.itfSaMController.IsPossibleExitState (eMode := E_BaseMachineMode.Washing)) THEN
			THIS^.itfSaMController.ChangeModeTo (eModeIn := E_BaseMachineMode.Washing);
		ELSE
			THIS^.EventSetActive (iNumber := 3);	//brak możlwiosći wejście do trybu w tym stanie 
		END_IF
	ELSE
		THIS^.EventSetActive (iNumber := 2);	//brak możliwości wyjścia w tym stanie z tego trybu
	END_IF
ELSE
	THIS^.EventSetActive (iNumber := 1);	//tryb docelowy wylaczony
END_IF
END_METHOD

METHOD FB_init : BOOL
VAR_INPUT
	bInitRetains : BOOL; // if TRUE, the retain variables are initialized (warm start / cold start)
	bInCopyCode : BOOL;  // if TRUE, the instance afterwards gets moved into the copy code (online change)
END_VAR
THIS^.SetText (eLocation := E_BaseLocation.pl, wsDescription := "Command change mode - Washing");
THIS^.SetText (eLocation := E_BaseLocation.en, wsDescription := "Command change mode - Washing");
THIS^.SetText (eLocation := E_BaseLocation.de, wsDescription := "Command change mode - Washing");
THIS^.SetName (stName := THIS^.GetTexts ());
END_METHOD

END_FUNCTION_BLOCK

// ---- POUs/04_CommandChangeMode/FB_CommandChangeDiagnostics.TcPOU
FUNCTION_BLOCK FB_CommandChangeDiagnostics EXTENDS FB_CommandChange IMPLEMENTS ITF_CommandChange
VAR

END_VAR

(*			
	RafalOS
	Rafał Osajda		03.11.2025		TC 4024.66
	Test czy można zmienić stan lub tryb i zwraca czy można i uruchamia zmianę
*)
METHOD PUBLIC Execute : BOOL
VAR_INPUT
	iNumberOfCommand	: INT;
END_VAR
IF (THIS^.itfSaMController.IsModeEnebles (eMode := E_BaseMachineMode.Diagnostics)) THEN
	IF (THIS^.itfSaMController.IsPossibleExitActiveState ()) THEN
		IF (THIS^.itfSaMController.IsPossibleExitState (eMode := E_BaseMachineMode.Diagnostics)) THEN
			THIS^.itfSaMController.ChangeModeTo (eModeIn := E_BaseMachineMode.Diagnostics);
		ELSE
			THIS^.EventSetActive (iNumber := 3);	//brak możlwiosći wejście do trybu w tym stanie 
		END_IF
	ELSE
		THIS^.EventSetActive (iNumber := 2);	//brak możliwości wyjścia w tym stanie z tego trybu
	END_IF
ELSE
	THIS^.EventSetActive (iNumber := 1);	//tryb docelowy wylaczony
END_IF
END_METHOD

METHOD FB_init : BOOL
VAR_INPUT
	bInitRetains : BOOL; // if TRUE, the retain variables are initialized (warm start / cold start)
	bInCopyCode : BOOL;  // if TRUE, the instance afterwards gets moved into the copy code (online change)
END_VAR
THIS^.SetText (eLocation := E_BaseLocation.pl, wsDescription := "Command change mode - Diagnostics");
THIS^.SetText (eLocation := E_BaseLocation.en, wsDescription := "Command change mode - Diagnostics");
THIS^.SetText (eLocation := E_BaseLocation.de, wsDescription := "Command change mode - Diagnostics");
THIS^.SetName (stName := THIS^.GetTexts ());
END_METHOD

END_FUNCTION_BLOCK

// ---- POUs/05_SaMElement/FB_SaMElement.TcPOU
FUNCTION_BLOCK ABSTRACT FB_SaMElement EXTENDS FB_BaseComponent IMPLEMENTS ITF_SaMElement
VAR
	bActive						: BOOL;				//informacja czy dany element jest aktywny 
	bIsEnabled					: BOOL;				//informacje czy dany element jest włączony
	bTypeActive					: BOOL;				//informacja czy stan jest stanem aktywnym końcówka ING 
END_VAR
VAR PERSISTENT
	ltWorkTime					: LTIME;				//czas pracy w danym stanie - trybie
END_VAR

METHOD public GetNextState : E_BaseMachineState
VAR_INPUT
END_VAR
END_METHOD

METHOD GetTime : LTIME
VAR_INPUT
END_VAR
GetTime := THIS^.ltWorkTime;
END_METHOD

METHOD PUBLIC IncrementTime
VAR_INPUT
	tInterval				: TIME := T#100MS;
END_VAR
THIS^.ltWorkTime			:= THIS^.ltWorkTime + TO_LTIME (tInterval);
END_METHOD

METHOD PUBLIC InvokeStateForTopElement : BOOL
VAR_INPUT
	itfTopElement		: ITF_BaseSaMStateMethod;
END_VAR
END_METHOD

METHOD PUBLIC IsActive : BOOL
VAR_INPUT
END_VAR
IsActive			:= THIS^.bActive;
END_METHOD

(*			
	RafalOS
	Rafał Osajda		03.11.2025		TC 4024.66
	Zwraca czy element jest właczony w systemie
*)
METHOD PUBLIC IsEnabled : BOOL
VAR_INPUT
END_VAR
IsEnabled			:= THIS^.bIsEnabled;
END_METHOD

METHOD PUBLIC IsStateTypeActive : BOOL
VAR_INPUT
END_VAR
IsStateTypeActive		:= THIS^.bTypeActive;
END_METHOD

METHOD PUBLIC ResetTime
VAR_INPUT
END_VAR
THIS^.ltWorkTime		:= LTIME#0MS;
END_METHOD

(*			
	RafalOS
	Rafał Osajda		03.11.2025		TC 4024.66
	Ustawia czy dane element jest aktywny
*)
METHOD PUBLIC SetActive
VAR_INPUT
	bIN			: BOOL;
END_VAR
THIS^.bActive	:= bIN;
END_METHOD

(*			
	RafalOS
	Rafał Osajda		03.11.2025		TC 4024.66
	Ustawie czy element jest włączony w systemie
*)
METHOD PUBLIC SetEnabled
VAR_INPUT
	bIN			: BOOL;
END_VAR
THIS^.bIsEnabled		:= bIN;
END_METHOD

END_FUNCTION_BLOCK

// ---- POUs/06_SaMElementStates/FB_SaMElementAborting.TcPOU
FUNCTION_BLOCK FB_SaMElementAborting EXTENDS FB_SaMElement
VAR
END_VAR

METHOD FB_init : BOOL
VAR_INPUT
	bInitRetains : BOOL; // if TRUE, the retain variables are initialized (warm start / cold start)
	bInCopyCode : BOOL;  // if TRUE, the instance afterwards gets moved into the copy code (online change)
END_VAR
THIS^.bTypeActive		:= TRUE;

THIS^.SetText (eLocation := E_BaseLocation.pl, wsDescription := "Przerywanie");
THIS^.SetText (eLocation := E_BaseLocation.en, wsDescription := "Aborting");
THIS^.SetText (eLocation := E_BaseLocation.de, wsDescription := "Abbruch");
THIS^.SetName (stName := THIS^.GetTexts ());
END_METHOD

METHOD public GetNextState : E_BaseMachineState
VAR_INPUT
END_VAR
GetNextState		:= E_BaseMachineState.Aborted;
END_METHOD

METHOD PUBLIC InvokeStateForTopElement : BOOL
VAR_INPUT
	itfTopElement		: ITF_BaseSaMStateMethod;
END_VAR
InvokeStateForTopElement	:= itfTopElement.SP_Aborting ();
END_METHOD

END_FUNCTION_BLOCK

// ---- POUs/06_SaMElementStates/FB_SaMElementStopped.TcPOU
FUNCTION_BLOCK FB_SaMElementStopped EXTENDS FB_SaMElement
VAR
END_VAR

METHOD FB_init : BOOL
VAR_INPUT
	bInitRetains : BOOL; // if TRUE, the retain variables are initialized (warm start / cold start)
	bInCopyCode : BOOL;  // if TRUE, the instance afterwards gets moved into the copy code (online change)
END_VAR
THIS^.bTypeActive		:= FALSE;

THIS^.SetText (eLocation := E_BaseLocation.pl, wsDescription := "Zatrzymany");
THIS^.SetText (eLocation := E_BaseLocation.en, wsDescription := "Stopped");
THIS^.SetText (eLocation := E_BaseLocation.de, wsDescription := "Gestoppt");
THIS^.SetName (stName := THIS^.GetTexts ());
END_METHOD

METHOD PUBLIC InvokeStateForTopElement : BOOL
VAR_INPUT
	itfTopElement		: ITF_BaseSaMStateMethod;
END_VAR
InvokeStateForTopElement	:= itfTopElement.SP_Stopped ();
END_METHOD

END_FUNCTION_BLOCK

// ---- POUs/06_SaMElementStates/FB_SaMElementResseting.TcPOU
FUNCTION_BLOCK FB_SaMElementResseting EXTENDS FB_SaMElement
VAR
END_VAR

METHOD FB_init : BOOL
VAR_INPUT
	bInitRetains : BOOL; // if TRUE, the retain variables are initialized (warm start / cold start)
	bInCopyCode : BOOL;  // if TRUE, the instance afterwards gets moved into the copy code (online change)
END_VAR
THIS^.bTypeActive		:= TRUE;

THIS^.SetText (eLocation := E_BaseLocation.pl, wsDescription := "Bazowanie");
THIS^.SetText (eLocation := E_BaseLocation.en, wsDescription := "Resetting");
THIS^.SetText (eLocation := E_BaseLocation.de, wsDescription := "Zurücksetzen");
THIS^.SetName (stName := THIS^.GetTexts ());
END_METHOD

METHOD public GetNextState : E_BaseMachineState
VAR_INPUT
END_VAR
GetNextState		:= E_BaseMachineState.Idle;
END_METHOD

METHOD PUBLIC InvokeStateForTopElement : BOOL
VAR_INPUT
	itfTopElement		: ITF_BaseSaMStateMethod;
END_VAR
InvokeStateForTopElement	:= itfTopElement.SP_Resetting ();
END_METHOD

END_FUNCTION_BLOCK

// ---- POUs/06_SaMElementStates/FB_SaMElementStarting.TcPOU
FUNCTION_BLOCK FB_SaMElementStarting EXTENDS FB_SaMElement
VAR
END_VAR

METHOD FB_init : BOOL
VAR_INPUT
	bInitRetains : BOOL; // if TRUE, the retain variables are initialized (warm start / cold start)
	bInCopyCode : BOOL;  // if TRUE, the instance afterwards gets moved into the copy code (online change)
END_VAR
THIS^.bTypeActive		:= TRUE;

THIS^.SetText (eLocation := E_BaseLocation.pl, wsDescription := "Uruchamianie");
THIS^.SetText (eLocation := E_BaseLocation.en, wsDescription := "Starting");
THIS^.SetText (eLocation := E_BaseLocation.de, wsDescription := "Beginnend");
THIS^.SetName (stName := THIS^.GetTexts ());
END_METHOD

METHOD public GetNextState : E_BaseMachineState
VAR_INPUT
END_VAR
GetNextState		:= E_BaseMachineState.Execute;
END_METHOD

METHOD PUBLIC InvokeStateForTopElement : BOOL
VAR_INPUT
	itfTopElement		: ITF_BaseSaMStateMethod;
END_VAR
InvokeStateForTopElement	:= itfTopElement.SP_Starting ();
END_METHOD

END_FUNCTION_BLOCK

// ---- POUs/06_SaMElementStates/FB_SaMElementSuspended.TcPOU
FUNCTION_BLOCK FB_SaMElementSuspended EXTENDS FB_SaMElement
VAR
END_VAR

METHOD FB_init : BOOL
VAR_INPUT
	bInitRetains : BOOL; // if TRUE, the retain variables are initialized (warm start / cold start)
	bInCopyCode : BOOL;  // if TRUE, the instance afterwards gets moved into the copy code (online change)
END_VAR
THIS^.bTypeActive		:= FALSE;

THIS^.SetText (eLocation := E_BaseLocation.pl, wsDescription := "Zawieszony");
THIS^.SetText (eLocation := E_BaseLocation.en, wsDescription := "Suspended");
THIS^.SetText (eLocation := E_BaseLocation.de, wsDescription := "Aussetzen");
THIS^.SetName (stName := THIS^.GetTexts ());
END_METHOD

METHOD PUBLIC InvokeStateForTopElement : BOOL
VAR_INPUT
	itfTopElement		: ITF_BaseSaMStateMethod;
END_VAR
InvokeStateForTopElement	:= itfTopElement.SP_Suspended ();
END_METHOD

END_FUNCTION_BLOCK

// ---- POUs/07_SaMElementModes/FB_SaMElementProduction.TcPOU
FUNCTION_BLOCK FB_SaMElementProduction EXTENDS FB_SaMElement
VAR
END_VAR

METHOD FB_init : BOOL
VAR_INPUT
	bInitRetains : BOOL; // if TRUE, the retain variables are initialized (warm start / cold start)
	bInCopyCode : BOOL;  // if TRUE, the instance afterwards gets moved into the copy code (online change)
END_VAR
THIS^.SetText (eLocation := E_BaseLocation.pl, wsDescription := "Produkcja");
THIS^.SetText (eLocation := E_BaseLocation.en, wsDescription := "Production");
THIS^.SetText (eLocation := E_BaseLocation.de, wsDescription := "Produktion");
THIS^.SetName (stName := THIS^.GetTexts ());
END_METHOD

END_FUNCTION_BLOCK

// ---- POUs/07_SaMElementModes/FB_SaMElementManual.TcPOU
FUNCTION_BLOCK FB_SaMElementManual EXTENDS FB_SaMElement
VAR
END_VAR

METHOD FB_init : BOOL
VAR_INPUT
	bInitRetains : BOOL; // if TRUE, the retain variables are initialized (warm start / cold start)
	bInCopyCode : BOOL;  // if TRUE, the instance afterwards gets moved into the copy code (online change)
END_VAR
THIS^.SetText (eLocation := E_BaseLocation.pl, wsDescription := "Ręczny");
THIS^.SetText (eLocation := E_BaseLocation.en, wsDescription := "Manual");
THIS^.SetText (eLocation := E_BaseLocation.de, wsDescription := "Handbuch");
THIS^.SetName (stName := THIS^.GetTexts ());
END_METHOD

END_FUNCTION_BLOCK

// ---- POUs/07_SaMElementModes/FB_SaMElementWashing.TcPOU
FUNCTION_BLOCK FB_SaMElementWashing EXTENDS FB_SaMElement
VAR
END_VAR

METHOD FB_init : BOOL
VAR_INPUT
	bInitRetains : BOOL; // if TRUE, the retain variables are initialized (warm start / cold start)
	bInCopyCode : BOOL;  // if TRUE, the instance afterwards gets moved into the copy code (online change)
END_VAR
THIS^.SetText (eLocation := E_BaseLocation.pl, wsDescription := "Mycie");
THIS^.SetText (eLocation := E_BaseLocation.en, wsDescription := "Washing");
THIS^.SetText (eLocation := E_BaseLocation.de, wsDescription := "Waschen");
THIS^.SetName (stName := THIS^.GetTexts ());
END_METHOD

END_FUNCTION_BLOCK
